KUKA KRL program: EPS_2_251719_MHSUMNERSTREET_A_20251210010858.src

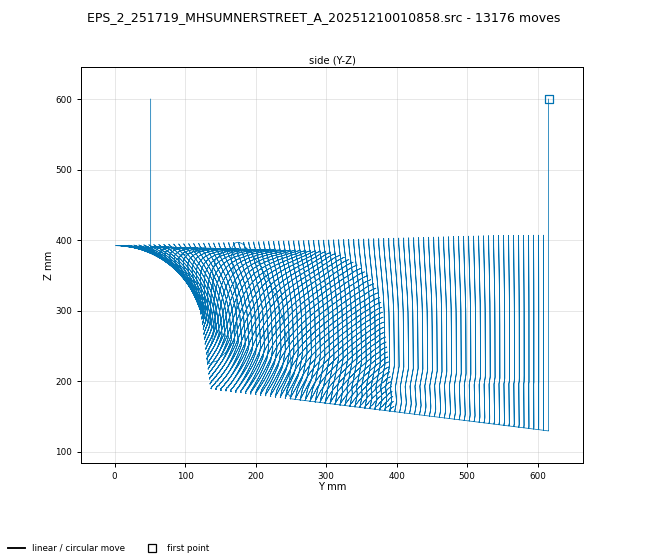
[picture p0: tool path of EPS_2_251719_MHSUMNERSTREET_A_20251210010858.src, 13176 of 13178 moves have a stored position in this frame; points joined in program order, loops and branches not executed]
&ACCESS RVP
&REL 4
&COMMENT QRS 19112012
&PARAM EDITMASK = *
DEF PART()
EXT BAS (BAS_COMMAND :IN,REAL :IN )
INT I
BAS (#INITMOV,0 )

;KUKA QRS Post kuka4.cps  Date:22-06-2017 !

File_ID=2952

QRS_PRE_INIT()

;Init var - Until changes are made in qrs_pre_init
Outlet_Square_prg=0
Inlet_1_Square_prg=0
Inlet_2_Square_prg=0
Inlet_3_Square_prg=0
Inlet_4_Square_prg=0
Inlet_5_Square_prg=0

Outlet_1={X 0.000, Y 546.330, Z 306.500, B 0.000, E1 0.000 }
Inlet_1={X 0.000, Y 567.240, Z 281.500, B 0.000, E1 180.000 }
Outlet_1_type=201
Inlet_1_type=0
;QRS#1=Sidecore dimensions
;QRS#2=200-8" PVC SDR 35
;QRS#3=DeadEnd 201
;QRS#4=
;QRS#5=
;QRS#6=
;QRS#7=
;QRS#8=
;QRS#9=12-08 PSX
;QRS#10=

;QRS#11=
;QRS#12=
;QRS#13=
;QRS#14=
;QRS#15=
;QRS#16=1220x127x686 2,25'
;QRS#17=EPS Height
;QRS#18=407
;QRS#19=*
;QRS#20= UPDATED VERSION 22-06-2017
;QRS#21=*
Outlet_Square=0100
Inlet_1_Square=00
Inlet_2_Square=0
Inlet_3_Square=0
Inlet_4_Square=0
Inlet_5_Square=0
Mill_Square=1
Outlet_Square_Prg=204
Inlet_1_Square_prg=0

QRS_INIT()

$ADVANCE=5

; T1
PTP {E1 173.614,E2 173.614}
PTP {X 0,Y 615.484,A -85,B 0,C 180,E1 173.614,E2 173.614,E3 0,E4 0,E5 0,E6 0}
QRS_SPEED_INIT()
LIN {X 0,Y 615.484,Z 600,A -85,B 0,C 180,E1 173.614,E2 173.614,E3 0,E4 0,E5 0,E6 0} C_VEL
LIN {X 0,Y 615.484,Z 139.376,A -85,B 0,C 180,E1 173.614,E2 173.614} C_VEL
LIN {X 0,Y 615.484,Z 131.194,A -85,B 0,C 180,E1 173.614,E2 173.614} C_VEL
LIN {X 0,Y 615.473,Z 129.194,A -85,B 0,C 180,E1 173.428,E2 173.428} C_VEL
LIN {X 0,Y 615.496,Z 129.181,A -85,B 0,C 180,E1 170.802,E2 170.802} C_VEL
LIN {X 0,Y 615.487,Z 129.196,A -85,B 0,C 180,E1 168.14,E2 168.14} C_VEL
LIN {X 0,Y 615.472,Z 129.19,A -85,B 0,C 180,E1 165.451,E2 165.451} C_VEL
LIN {X 0,Y 615.485,Z 129.186,A -85,B 0,C 180,E1 162.73,E2 162.73} C_VEL
LIN {X 0,Y 615.482,Z 129.198,A -85,B 0,C 180,E1 159.967,E2 159.967} C_VEL
LIN {X 0,Y 615.487,Z 129.183,A -85,B 0,C 180,E1 157.156,E2 157.156} C_VEL
LIN {X 0,Y 615.498,Z 129.2,A -85,B 0,C 180,E1 154.285,E2 154.285} C_VEL
LIN {X 0,Y 615.486,Z 129.183,A -85,B 0,C 180,E1 151.342,E2 151.342} C_VEL
LIN {X 0,Y 615.48,Z 129.19,A -85,B 0,C 180,E1 148.914,E2 148.914} C_VEL
LIN {X 0,Y 615.496,Z 129.199,A -85,B 0,C 180,E1 146.464,E2 146.464} C_VEL
LIN {X 0,Y 615.483,Z 129.184,A -85,B 0,C 180,E1 143.575,E2 143.575} C_VEL
LIN {X 0,Y 615.484,Z 129.194,A -85,B 0,C 180,E1 140.938,E2 140.938} C_VEL
LIN {X 0,Y 615.485,Z 129.197,A -85,B 0,C 180,E1 138.527,E2 138.527} C_VEL
LIN {X 0,Y 615.49,Z 129.182,A -85,B 0,C 180,E1 135.851,E2 135.851} C_VEL
LIN {X 0,Y 615.488,Z 129.196,A -85,B 0,C 180,E1 133.048,E2 133.048} C_VEL
LIN {X 0,Y 615.479,Z 129.194,A -85,B 0,C 180,E1 130.607,E2 130.607} C_VEL
LIN {X 0,Y 615.482,Z 129.184,A -85,B 0,C 180,E1 128.012,E2 128.012} C_VEL
LIN {X 0,Y 615.481,Z 129.188,A -85,B 0,C 180,E1 125.616,E2 125.616} C_VEL
LIN {X 0,Y 615.484,Z 129.199,A -85,B 0,C 180,E1 123.236,E2 123.236} C_VEL
LIN {X 0,Y 615.478,Z 129.196,A -85,B 0,C 180,E1 120.92,E2 120.92} C_VEL
LIN {X 0,Y 615.483,Z 129.185,A -85,B 0,C 180,E1 118.45,E2 118.45} C_VEL
LIN {X 0,Y 615.484,Z 129.195,A -85,B 0,C 180,E1 115.569,E2 115.569} C_VEL
LIN {X 0,Y 615.475,Z 129.19,A -85,B 0,C 180,E1 112.845,E2 112.845} C_VEL
LIN {X 0,Y 615.49,Z 129.183,A -85,B 0,C 180,E1 110.559,E2 110.559} C_VEL
LIN {X 0,Y 615.479,Z 129.191,A -85,B 0,C 180,E1 107.957,E2 107.957} C_VEL
LIN {X 0,Y 615.479,Z 129.193,A -85,B 0,C 180,E1 105.226,E2 105.226} C_VEL
LIN {X 0,Y 615.491,Z 129.182,A -85,B 0,C 180,E1 102.53,E2 102.53} C_VEL
LIN {X 0,Y 615.491,Z 129.198,A -85,B 0,C 180,E1 99.862,E2 99.862} C_VEL
LIN {X 0,Y 615.477,Z 129.189,A -85,B 0,C 180,E1 97.216,E2 97.216} C_VEL
LIN {X 0,Y 615.482,Z 129.186,A -85,B 0,C 180,E1 94.585,E2 94.585} C_VEL
LIN {X 0,Y 615.499,Z 129.2,A -85,B 0,C 180,E1 91.963,E2 91.963} C_VEL
LIN {X 0,Y 615.481,Z 129.187,A -85,B 0,C 180,E1 89.346,E2 89.346} C_VEL
LIN {X 0,Y 615.479,Z 129.187,A -85,B 0,C 180,E1 86.727,E2 86.727} C_VEL
LIN {X 0,Y 615.496,Z 129.199,A -85,B 0,C 180,E1 84.102,E2 84.102} C_VEL
LIN {X 0,Y 615.485,Z 129.185,A -85,B 0,C 180,E1 81.463,E2 81.463} C_VEL
LIN {X 0,Y 615.477,Z 129.19,A -85,B 0,C 180,E1 78.807,E2 78.807} C_VEL
LIN {X 0,Y 615.482,Z 129.194,A -85,B 0,C 180,E1 76.067,E2 76.067} C_VEL
LIN {X 0,Y 615.487,Z 129.183,A -85,B 0,C 180,E1 73.414,E2 73.414} C_VEL
LIN {X 0,Y 615.484,Z 129.198,A -85,B 0,C 180,E1 70.662,E2 70.662} C_VEL
LIN {X 0,Y 615.479,Z 129.186,A -85,B 0,C 180,E1 67.864,E2 67.864} C_VEL
LIN {X 0,Y 615.488,Z 129.183,A -85,B 0,C 180,E1 65.728,E2 65.728} C_VEL
LIN {X 0,Y 615.484,Z 129.2,A -85,B 0,C 180,E1 62.823,E2 62.823} C_VEL
LIN {X 0,Y 615.499,Z 129.18,A -85,B 0,C 180,E1 59.841,E2 59.841} C_VEL
LIN {X 0,Y 615.478,Z 129.187,A -85,B 0,C 180,E1 57.542,E2 57.542} C_VEL
LIN {X 0,Y 615.477,Z 129.196,A -85,B 0,C 180,E1 55.185,E2 55.185} C_VEL
LIN {X 0,Y 615.486,Z 129.195,A -85,B 0,C 180,E1 52.758,E2 52.758} C_VEL
LIN {X 0,Y 615.485,Z 129.184,A -85,B 0,C 180,E1 49.911,E2 49.911} C_VEL
LIN {X 0,Y 615.488,Z 129.196,A -85,B 0,C 180,E1 46.952,E2 46.952} C_VEL
LIN {X 0,Y 615.481,Z 129.185,A -85,B 0,C 180,E1 43.997,E2 43.997} C_VEL
LIN {X 0,Y 615.485,Z 129.197,A -85,B 0,C 180,E1 41.473,E2 41.473} C_VEL
LIN {X 0,Y 615.481,Z 129.191,A -85,B 0,C 180,E1 38.904,E2 38.904} C_VEL
LIN {X 0,Y 615.483,Z 129.184,A -85,B 0,C 180,E1 36.425,E2 36.425} C_VEL
LIN {X 0,Y 615.496,Z 129.199,A -85,B 0,C 180,E1 33.536,E2 33.536} C_VEL
LIN {X 0,Y 615.484,Z 129.186,A -85,B 0,C 180,E1 30.919,E2 30.919} C_VEL
LIN {X 0,Y 615.48,Z 129.185,A -85,B 0,C 180,E1 28.45,E2 28.45} C_VEL
LIN {X 0,Y 615.488,Z 129.198,A -85,B 0,C 180,E1 25.57,E2 25.57} C_VEL
LIN {X 0,Y 615.487,Z 129.183,A -85,B 0,C 180,E1 22.844,E2 22.844} C_VEL
LIN {X 0,Y 615.482,Z 129.198,A -85,B 0,C 180,E1 20.033,E2 20.033} C_VEL
LIN {X 0,Y 615.481,Z 129.187,A -85,B 0,C 180,E1 17.27,E2 17.27} C_VEL
LIN {X 0,Y 615.472,Z 129.19,A -85,B 0,C 180,E1 14.549,E2 14.549} C_VEL
LIN {X 0,Y 615.487,Z 129.196,A -85,B 0,C 180,E1 11.86,E2 11.86} C_VEL
LIN {X 0,Y 615.496,Z 129.181,A -85,B 0,C 180,E1 9.198,E2 9.198} C_VEL
LIN {X 0,Y 615.474,Z 129.195,A -85,B 0,C 180,E1 6.556,E2 6.556} C_VEL
LIN {X 0,Y 615.484,Z 129.192,A -85,B 0,C 180,E1 3.928,E2 3.928} C_VEL
LIN {X 0,Y 615.487,Z 129.183,A -85,B 0,C 180,E1 1.308,E2 1.308} C_VEL
LIN {X 0,Y 615.479,Z 129.195,A -85,B 0,C 180,E1 -1.309,E2 -1.309} C_VEL
LIN {X 0,Y 615.483,Z 129.191,A -85,B 0,C 180,E1 -3.929,E2 -3.929} C_VEL
LIN {X 0,Y 615.48,Z 129.185,A -85,B 0,C 180,E1 -6.577,E2 -6.577} C_VEL
LIN {X 0,Y 615.485,Z 129.197,A -85,B 0,C 180,E1 -9.199,E2 -9.199} C_VEL
LIN {X 0,Y 615.485,Z 129.187,A -85,B 0,C 180,E1 -11.861,E2 -11.861} C_VEL
LIN {X 0,Y 615.473,Z 129.188,A -85,B 0,C 180,E1 -14.55,E2 -14.55} C_VEL
LIN {X 0,Y 615.491,Z 129.198,A -85,B 0,C 180,E1 -17.271,E2 -17.271} C_VEL
LIN {X 0,Y 615.486,Z 129.183,A -85,B 0,C 180,E1 -20.033,E2 -20.033} C_VEL
LIN {X 0,Y 615.48,Z 129.199,A -85,B 0,C 180,E1 -22.845,E2 -22.845} C_VEL
LIN {X 0,Y 615.495,Z 129.182,A -85,B 0,C 180,E1 -25.716,E2 -25.716} C_VEL
LIN {X 0,Y 615.473,Z 129.193,A -85,B 0,C 180,E1 -28.449,E2 -28.449} C_VEL
LIN {X 0,Y 615.486,Z 129.193,A -85,B 0,C 180,E1 -31.087,E2 -31.087} C_VEL
LIN {X 0,Y 615.471,Z 129.188,A -85,B 0,C 180,E1 -34.023,E2 -34.023} C_VEL
LIN {X 0,Y 615.48,Z 129.197,A -85,B 0,C 180,E1 -36.426,E2 -36.426} C_VEL
LIN {X 0,Y 615.485,Z 129.189,A -85,B 0,C 180,E1 -39.063,E2 -39.063} C_VEL
LIN {X 0,Y 615.484,Z 129.184,A -85,B 0,C 180,E1 -41.474,E2 -41.474} C_VEL
LIN {X 0,Y 615.475,Z 129.196,A -85,B 0,C 180,E1 -44.151,E2 -44.151} C_VEL
LIN {X 0,Y 615.486,Z 129.187,A -85,B 0,C 180,E1 -46.953,E2 -46.953} C_VEL
LIN {X 0,Y 615.477,Z 129.185,A -85,B 0,C 180,E1 -49.393,E2 -49.393} C_VEL
LIN {X 0,Y 615.478,Z 129.196,A -85,B 0,C 180,E1 -51.99,E2 -51.99} C_VEL
LIN {X 0,Y 615.489,Z 129.195,A -85,B 0,C 180,E1 -54.385,E2 -54.385} C_VEL
LIN {X 0,Y 615.486,Z 129.186,A -85,B 0,C 180,E1 -56.764,E2 -56.764} C_VEL
LIN {X 0,Y 615.479,Z 129.185,A -85,B 0,C 180,E1 -59.08,E2 -59.08} C_VEL
LIN {X 0,Y 615.471,Z 129.193,A -85,B 0,C 180,E1 -61.553,E2 -61.553} C_VEL
LIN {X 0,Y 615.487,Z 129.188,A -85,B 0,C 180,E1 -64.432,E2 -64.432} C_VEL
LIN {X 0,Y 615.497,Z 129.361,A -85,B 0,C 180,E1 -65.958,E2 -65.958} C_VEL
LIN {X 0,Y 615.498,Z 144.439,A -85,B 0,C 180,E1 -68.569,E2 -68.569} C_VEL
LIN {X 0,Y 615.482,Z 161.223,A -85,B 0,C 180,E1 -71.398,E2 -71.398} C_VEL
LIN {X 0,Y 615.496,Z 178.498,A -85,B 0,C 180,E1 -74.265,E2 -74.265} C_VEL
LIN {X 0,Y 615.469,Z 195.732,A -85,B 0,C 180,E1 -77.071,E2 -77.071} C_VEL
LIN {X 0,Y 615.464,Z 197.255,A -85,B 0,C 180,E1 -77.155,E2 -77.155} C_VEL
LIN {X 0,Y 615.498,Z 302.835,A -85,B 0,C 180,E1 -78.411,E2 -78.411} C_VEL
LIN {X 0,Y 615.499,Z 315.346,A -85,B 0,C 180,E1 -78.682,E2 -78.682} C_VEL
LIN {X 0,Y 615.496,Z 328.502,A -85,B 0,C 180,E1 -79.109,E2 -79.109} C_VEL
LIN {X 0,Y 615.487,Z 340.479,A -85,B 0,C 180,E1 -79.64,E2 -79.64} C_VEL
LIN {X 0,Y 615.493,Z 351.996,A -85,B 0,C 180,E1 -80.304,E2 -80.304} C_VEL
LIN {X 0,Y 615.499,Z 362.342,A -85,B 0,C 180,E1 -81.05,E2 -81.05} C_VEL
LIN {X 0,Y 615.497,Z 370.813,A -85,B 0,C 180,E1 -81.794,E2 -81.794} C_VEL
LIN {X 0,Y 615.498,Z 378.607,A -85,B 0,C 180,E1 -82.62,E2 -82.62} C_VEL
LIN {X 0,Y 615.496,Z 386.203,A -85,B 0,C 180,E1 -83.608,E2 -83.608} C_VEL
LIN {X 0,Y 615.498,Z 393.205,A -85,B 0,C 180,E1 -84.759,E2 -84.759} C_VEL
LIN {X 0,Y 615.493,Z 397.852,A -85,B 0,C 180,E1 -85.744,E2 -85.744} C_VEL
LIN {X 0,Y 615.494,Z 401.399,A -85,B 0,C 180,E1 -86.727,E2 -86.727} C_VEL
LIN {X 0,Y 615.497,Z 403.233,A -85,B 0,C 180,E1 -87.382,E2 -87.382} C_VEL
LIN {X 0,Y 615.5,Z 404.607,A -85,B 0,C 180,E1 -88.037,E2 -88.037} C_VEL
LIN {X 0,Y 615.496,Z 406.173,A -85,B 0,C 180,E1 -89.346,E2 -89.346} C_VEL
LIN {X 0,Y 615.494,Z 406.389,A -85,B 0,C 180,E1 -90,E2 -90} C_VEL
LIN {X 0,Y 615.495,Z 405.58,A -85,B 0,C 180,E1 -91.309,E2 -91.309} C_VEL
LIN {X 0,Y 615.5,Z 404.607,A -85,B 0,C 180,E1 -91.963,E2 -91.963} C_VEL
LIN {X 0,Y 615.497,Z 403.233,A -85,B 0,C 180,E1 -92.618,E2 -92.618} C_VEL
LIN {X 0,Y 615.496,Z 400.35,A -85,B 0,C 180,E1 -93.601,E2 -93.601} C_VEL
LIN {X 0,Y 615.498,Z 396.442,A -85,B 0,C 180,E1 -94.584,E2 -94.584} C_VEL
LIN {X 0,Y 615.499,Z 391.405,A -85,B 0,C 180,E1 -95.57,E2 -95.57} C_VEL
LIN {X 0,Y 615.497,Z 384.87,A -85,B 0,C 180,E1 -96.583,E2 -96.583} C_VEL
LIN {X 0,Y 615.497,Z 377.134,A -85,B 0,C 180,E1 -97.545,E2 -97.545} C_VEL
LIN {X 0,Y 615.498,Z 369.046,A -85,B 0,C 180,E1 -98.371,E2 -98.371} C_VEL
LIN {X 0,Y 615.499,Z 359.169,A -85,B 0,C 180,E1 -99.199,E2 -99.199} C_VEL
LIN {X 0,Y 615.487,Z 347.983,A -85,B 0,C 180,E1 -99.945,E2 -99.945} C_VEL
LIN {X 0,Y 615.492,Z 337.024,A -85,B 0,C 180,E1 -100.527,E2 -100.527} C_VEL
LIN {X 0,Y 615.499,Z 324.42,A -85,B 0,C 180,E1 -101.042,E2 -101.042} C_VEL
LIN {X 0,Y 615.499,Z 312.068,A -85,B 0,C 180,E1 -101.401,E2 -101.401} C_VEL
LIN {X 0,Y 615.499,Z 298.472,A -85,B 0,C 180,E1 -101.652,E2 -101.652} C_VEL
LIN {X 0,Y 615.465,Z 196.548,A -85,B 0,C 180,E1 -102.866,E2 -102.866} C_VEL
LIN {X 0,Y 615.478,Z 194.988,A -85,B 0,C 180,E1 -103.033,E2 -103.033} C_VEL
LIN {X 0,Y 615.493,Z 177.465,A -85,B 0,C 180,E1 -105.905,E2 -105.905} C_VEL
LIN {X 0,Y 615.49,Z 159.928,A -85,B 0,C 180,E1 -108.818,E2 -108.818} C_VEL
LIN {X 0,Y 615.484,Z 143.406,A -85,B 0,C 180,E1 -111.608,E2 -111.608} C_VEL
LIN {X 0,Y 615.497,Z 129.361,A -85,B 0,C 180,E1 -114.042,E2 -114.042} C_VEL
LIN {X 0,Y 615.47,Z 129.194,A -85,B 0,C 180,E1 -116.445,E2 -116.445} C_VEL
LIN {X 0,Y 615.469,Z 129.19,A -85,B 0,C 180,E1 -118.659,E2 -118.659} C_VEL
LIN {X 0,Y 615.485,Z 129.184,A -85,B 0,C 180,E1 -121.085,E2 -121.085} C_VEL
LIN {X 0,Y 615.483,Z 129.198,A -85,B 0,C 180,E1 -124.022,E2 -124.022} C_VEL
LIN {X 0,Y 615.488,Z 129.183,A -85,B 0,C 180,E1 -126.936,E2 -126.936} C_VEL
LIN {X 0,Y 615.496,Z 129.199,A -85,B 0,C 180,E1 -129.749,E2 -129.749} C_VEL
LIN {X 0,Y 615.47,Z 129.188,A -85,B 0,C 180,E1 -132.354,E2 -132.354} C_VEL
LIN {X 0,Y 615.486,Z 129.188,A -85,B 0,C 180,E1 -135.068,E2 -135.068} C_VEL
LIN {X 0,Y 615.482,Z 129.199,A -85,B 0,C 180,E1 -137.646,E2 -137.646} C_VEL
LIN {X 0,Y 615.474,Z 129.186,A -85,B 0,C 180,E1 -140.248,E2 -140.248} C_VEL
LIN {X 0,Y 615.486,Z 129.193,A -85,B 0,C 180,E1 -143.063,E2 -143.063} C_VEL
LIN {X 0,Y 615.491,Z 129.202,A -85,B 0,C 180,E1 -145.298,E2 -145.298} C_VEL
LIN {X 0,Y 615.472,Z 129.193,A -85,B 0,C 180,E1 -147.671,E2 -147.671} C_VEL
LIN {X 0,Y 615.487,Z 129.183,A -85,B 0,C 180,E1 -150.204,E2 -150.204} C_VEL
LIN {X 0,Y 615.491,Z 129.197,A -85,B 0,C 180,E1 -152.953,E2 -152.953} C_VEL
LIN {X 0,Y 615.472,Z 129.188,A -85,B 0,C 180,E1 -155.727,E2 -155.727} C_VEL
LIN {X 0,Y 615.484,Z 129.191,A -85,B 0,C 180,E1 -158.568,E2 -158.568} C_VEL
LIN {X 0,Y 615.471,Z 129.191,A -85,B 0,C 180,E1 -161.398,E2 -161.398} C_VEL
LIN {X 0,Y 615.491,Z 129.184,A -85,B 0,C 180,E1 -164.095,E2 -164.095} C_VEL
LIN {X 0,Y 615.494,Z 129.199,A -85,B 0,C 180,E1 -166.799,E2 -166.799} C_VEL
LIN {X 0,Y 615.477,Z 129.186,A -85,B 0,C 180,E1 -169.473,E2 -169.473} C_VEL
LIN {X 0,Y 615.483,Z 129.19,A -85,B 0,C 180,E1 -172.124,E2 -172.124} C_VEL
LIN {X 0,Y 615.481,Z 129.196,A -85,B 0,C 180,E1 -174.758,E2 -174.758} C_VEL
LIN {X 0,Y 615.484,Z 129.184,A -85,B 0,C 180,E1 -177.382,E2 -177.382} C_VEL
LIN {X 0,Y 615.483,Z 129.192,A -85,B 0,C 180,E1 -180,E2 -180} C_VEL
LIN {X 0,Y 615.478,Z 129.195,A -85,B 0,C 180,E1 -182.618,E2 -182.618} C_VEL
LIN {X 0,Y 615.49,Z 129.182,A -85,B 0,C 180,E1 -185.241,E2 -185.241} C_VEL
LIN {X 0,Y 615.473,Z 129.194,A -85,B 0,C 180,E1 -186.572,E2 -186.572} C_VEL
LIN {X 0,Y 614.807,Z 129.333,A -85,B 0,C 180,E1 -187.118,E2 -187.118} C_VEL
LIN {X 0,Y 611.985,Z 129.755,A -85,B 0,C 180,E1 -188.004,E2 -188.004} C_VEL
LIN {X 0,Y 609.596,Z 130.06,A -85,B 0,C 180,E1 -188.717,E2 -188.717} C_VEL
LIN {X 0,Y 608.556,Z 130.176,A -85,B 0,C 180,E1 -189.266,E2 -189.266} C_VEL
LIN {X 0,Y 608.464,Z 130.187,A -85,B 0,C 180,E1 -189.452,E2 -189.452} C_VEL
LIN {X 0,Y 608.46,Z 130.196,A -85,B 0,C 180,E1 -191.999,E2 -191.999} C_VEL
LIN {X 0,Y 608.467,Z 130.187,A -85,B 0,C 180,E1 -194.72,E2 -194.72} C_VEL
LIN {X 0,Y 608.454,Z 130.191,A -85,B 0,C 180,E1 -197.476,E2 -197.476} C_VEL
LIN {X 0,Y 608.456,Z 130.191,A -85,B 0,C 180,E1 -200.274,E2 -200.274} C_VEL
LIN {X 0,Y 608.451,Z 130.189,A -85,B 0,C 180,E1 -203.124,E2 -203.124} C_VEL
LIN {X 0,Y 608.449,Z 130.192,A -85,B 0,C 180,E1 -206.035,E2 -206.035} C_VEL
LIN {X 0,Y 608.469,Z 130.185,A -85,B 0,C 180,E1 -208.62,E2 -208.62} C_VEL
LIN {X 0,Y 608.472,Z 130.192,A -85,B 0,C 180,E1 -211.316,E2 -211.316} C_VEL
LIN {X 0,Y 608.475,Z 130.191,A -85,B 0,C 180,E1 -213.736,E2 -213.736} C_VEL
LIN {X 0,Y 608.471,Z 130.186,A -85,B 0,C 180,E1 -216.09,E2 -216.09} C_VEL
LIN {X 0,Y 608.463,Z 130.187,A -85,B 0,C 180,E1 -218.588,E2 -218.588} C_VEL
LIN {X 0,Y 608.46,Z 130.196,A -85,B 0,C 180,E1 -221.343,E2 -221.343} C_VEL
LIN {X 0,Y 608.458,Z 130.187,A -85,B 0,C 180,E1 -224.265,E2 -224.265} C_VEL
LIN {X 0,Y 608.453,Z 130.196,A -85,B 0,C 180,E1 -227.041,E2 -227.041} C_VEL
LIN {X 0,Y 608.447,Z 130.19,A -85,B 0,C 180,E1 -229.697,E2 -229.697} C_VEL
LIN {X 0,Y 608.467,Z 130.187,A -85,B 0,C 180,E1 -232.254,E2 -232.254} C_VEL
LIN {X 0,Y 608.473,Z 130.192,A -85,B 0,C 180,E1 -235.091,E2 -235.091} C_VEL
LIN {X 0,Y 608.463,Z 130.186,A -85,B 0,C 180,E1 -237.906,E2 -237.906} C_VEL
LIN {X 0,Y 608.465,Z 130.188,A -85,B 0,C 180,E1 -240.221,E2 -240.221} C_VEL
LIN {X 0,Y 608.477,Z 130.194,A -85,B 0,C 180,E1 -242.792,E2 -242.792} C_VEL
LIN {X 0,Y 608.452,Z 130.188,A -85,B 0,C 180,E1 -245.429,E2 -245.429} C_VEL
LIN {X 0,Y 608.473,Z 130.191,A -85,B 0,C 180,E1 -248.309,E2 -248.309} C_VEL
LIN {X 0,Y 608.471,Z 130.186,A -85,B 0,C 180,E1 -251.283,E2 -251.283} C_VEL
LIN {X 0,Y 608.458,Z 130.19,A -85,B 0,C 180,E1 -253.906,E2 -253.906} C_VEL
LIN {X 0,Y 608.456,Z 130.193,A -85,B 0,C 180,E1 -256.644,E2 -256.644} C_VEL
LIN {X 0,Y 608.464,Z 130.186,A -85,B 0,C 180,E1 -259.35,E2 -259.35} C_VEL
LIN {X 0,Y 608.477,Z 130.192,A -85,B 0,C 180,E1 -262.033,E2 -262.033} C_VEL
LIN {X 0,Y 608.46,Z 130.189,A -85,B 0,C 180,E1 -264.698,E2 -264.698} C_VEL
LIN {X 0,Y 608.472,Z 130.186,A -85,B 0,C 180,E1 -267.352,E2 -267.352} C_VEL
LIN {X 0,Y 608.477,Z 130.195,A -85,B 0,C 180,E1 -270,E2 -270} C_VEL
LIN {X 0,Y 608.472,Z 130.186,A -85,B 0,C 180,E1 -272.648,E2 -272.648} C_VEL
LIN {X 0,Y 608.46,Z 130.189,A -85,B 0,C 180,E1 -275.302,E2 -275.302} C_VEL
LIN {X 0,Y 608.477,Z 130.192,A -85,B 0,C 180,E1 -277.967,E2 -277.967} C_VEL
LIN {X 0,Y 608.467,Z 130.186,A -85,B 0,C 180,E1 -280.957,E2 -280.957} C_VEL
LIN {X 0,Y 608.455,Z 130.193,A -85,B 0,C 180,E1 -283.356,E2 -283.356} C_VEL
LIN {X 0,Y 608.456,Z 130.19,A -85,B 0,C 180,E1 -286.094,E2 -286.094} C_VEL
LIN {X 0,Y 608.455,Z 130.189,A -85,B 0,C 180,E1 -288.869,E2 -288.869} C_VEL
LIN {X 0,Y 608.473,Z 130.191,A -85,B 0,C 180,E1 -291.691,E2 -291.691} C_VEL
LIN {X 0,Y 608.45,Z 130.188,A -85,B 0,C 180,E1 -294.571,E2 -294.571} C_VEL
LIN {X 0,Y 608.477,Z 130.194,A -85,B 0,C 180,E1 -297.208,E2 -297.208} C_VEL
LIN {X 0,Y 608.468,Z 130.186,A -85,B 0,C 180,E1 -299.972,E2 -299.972} C_VEL
LIN {X 0,Y 608.454,Z 130.189,A -85,B 0,C 180,E1 -302.522,E2 -302.522} C_VEL
LIN {X 0,Y 608.437,Z 130.196,A -85,B 0,C 180,E1 -305.278,E2 -305.278} C_VEL
LIN {X 0,Y 608.468,Z 130.186,A -85,B 0,C 180,E1 -307.746,E2 -307.746} C_VEL
LIN {X 0,Y 608.448,Z 130.19,A -85,B 0,C 180,E1 -310.329,E2 -310.329} C_VEL
LIN {X 0,Y 608.453,Z 130.196,A -85,B 0,C 180,E1 -312.959,E2 -312.959} C_VEL
LIN {X 0,Y 608.458,Z 130.187,A -85,B 0,C 180,E1 -315.735,E2 -315.735} C_VEL
LIN {X 0,Y 608.46,Z 130.196,A -85,B 0,C 180,E1 -318.657,E2 -318.657} C_VEL
LIN {X 0,Y 608.463,Z 130.187,A -85,B 0,C 180,E1 -321.412,E2 -321.412} C_VEL
LIN {X 0,Y 608.471,Z 130.187,A -85,B 0,C 180,E1 -323.951,E2 -323.951} C_VEL
LIN {X 0,Y 608.467,Z 130.193,A -85,B 0,C 180,E1 -326.33,E2 -326.33} C_VEL
LIN {X 0,Y 608.472,Z 130.191,A -85,B 0,C 180,E1 -328.727,E2 -328.727} C_VEL
LIN {X 0,Y 608.471,Z 130.185,A -85,B 0,C 180,E1 -331.379,E2 -331.379} C_VEL
LIN {X 0,Y 608.477,Z 130.195,A -85,B 0,C 180,E1 -334.277,E2 -334.277} C_VEL
LIN {X 0,Y 608.451,Z 130.189,A -85,B 0,C 180,E1 -336.876,E2 -336.876} C_VEL
LIN {X 0,Y 608.456,Z 130.191,A -85,B 0,C 180,E1 -339.726,E2 -339.726} C_VEL
LIN {X 0,Y 608.452,Z 130.191,A -85,B 0,C 180,E1 -342.524,E2 -342.524} C_VEL
LIN {X 0,Y 608.467,Z 130.187,A -85,B 0,C 180,E1 -345.28,E2 -345.28} C_VEL
LIN {X 0,Y 608.46,Z 130.196,A -85,B 0,C 180,E1 -348.001,E2 -348.001} C_VEL
LIN {X 0,Y 608.477,Z 130.184,A -85,B 0,C 180,E1 -350.695,E2 -350.695} C_VEL
LIN {X 0,Y 608.452,Z 130.191,A -85,B 0,C 180,E1 -353.385,E2 -353.385} C_VEL
LIN {X 0,Y 608.452,Z 130.193,A -85,B 0,C 180,E1 -356.026,E2 -356.026} C_VEL
LIN {X 0,Y 608.47,Z 130.185,A -85,B 0,C 180,E1 -358.677,E2 -358.677} C_VEL
LIN {X 0,Y 608.463,Z 130.192,A -85,B 0,C 180,E1 -361.324,E2 -361.324} C_VEL
LIN {X 0,Y 608.452,Z 130.191,A -85,B 0,C 180,E1 -363.974,E2 -363.974} C_VEL
LIN {X 0,Y 608.474,Z 130.185,A -85,B 0,C 180,E1 -366.633,E2 -366.633} C_VEL
LIN {X 0,Y 608.469,Z 130.195,A -85,B 0,C 180,E1 -369.306,E2 -369.306} C_VEL
LIN {X 0,Y 608.458,Z 130.188,A -85,B 0,C 180,E1 -372,E2 -372} C_VEL
LIN {X 0,Y 608.467,Z 130.188,A -85,B 0,C 180,E1 -374.721,E2 -374.721} C_VEL
LIN {X 0,Y 608.457,Z 130.192,A -85,B 0,C 180,E1 -377.477,E2 -377.477} C_VEL
LIN {X 0,Y 608.456,Z 130.187,A -85,B 0,C 180,E1 -380.275,E2 -380.275} C_VEL
LIN {X 0,Y 608.456,Z 130.189,A -85,B 0,C 180,E1 -382.477,E2 -382.477} C_VEL
LIN {X 0,Y 608.453,Z 130.192,A -85,B 0,C 180,E1 -385.301,E2 -385.301} C_VEL
LIN {X 0,Y 608.448,Z 130.189,A -85,B 0,C 180,E1 -387.518,E2 -387.518} C_VEL
LIN {X 0,Y 608.463,Z 130.186,A -85,B 0,C 180,E1 -389.972,E2 -389.972} C_VEL
LIN {X 0,Y 608.454,Z 130.194,A -85,B 0,C 180,E1 -392.522,E2 -392.522} C_VEL
LIN {X 0,Y 608.448,Z 130.19,A -85,B 0,C 180,E1 -395.278,E2 -395.278} C_VEL
LIN {X 0,Y 608.46,Z 130.187,A -85,B 0,C 180,E1 -397.747,E2 -397.747} C_VEL
LIN {X 0,Y 608.445,Z 130.195,A -85,B 0,C 180,E1 -400.329,E2 -400.329} C_VEL
LIN {X 0,Y 608.481,Z 130.184,A -85,B 0,C 180,E1 -403.311,E2 -403.311} C_VEL
LIN {X 0,Y 608.46,Z 130.192,A -85,B 0,C 180,E1 -406.13,E2 -406.13} C_VEL
LIN {X 0,Y 608.458,Z 130.189,A -85,B 0,C 180,E1 -408.824,E2 -408.824} C_VEL
LIN {X 0,Y 608.47,Z 130.186,A -85,B 0,C 180,E1 -411.413,E2 -411.413} C_VEL
LIN {X 0,Y 608.447,Z 130.195,A -85,B 0,C 180,E1 -413.955,E2 -413.955} C_VEL
LIN {X 0,Y 608.467,Z 130.193,A -85,B 0,C 180,E1 -416.33,E2 -416.33} C_VEL
LIN {X 0,Y 608.479,Z 130.186,A -85,B 0,C 180,E1 -418.728,E2 -418.728} C_VEL
LIN {X 0,Y 608.459,Z 130.188,A -85,B 0,C 180,E1 -421.383,E2 -421.383} C_VEL
LIN {X 0,Y 608.44,Z 130.2,A -85,B 0,C 180,E1 -423.965,E2 -423.965} C_VEL
LIN {X 0,Y 608.496,Z 130.349,A -85,B 0,C 180,E1 -425.844,E2 -425.844} C_VEL
LIN {X 0,Y 608.531,Z 144.463,A -85,B 0,C 180,E1 -428.311,E2 -428.311} C_VEL
LIN {X 0,Y 608.51,Z 161.02,A -85,B 0,C 180,E1 -431.132,E2 -431.132} C_VEL
LIN {X 0,Y 608.483,Z 177.577,A -85,B 0,C 180,E1 -433.907,E2 -433.907} C_VEL
LIN {X 0,Y 608.481,Z 194.133,A -85,B 0,C 180,E1 -436.644,E2 -436.644} C_VEL
LIN {X 0,Y 608.461,Z 196.249,A -85,B 0,C 180,E1 -436.962,E2 -436.962} C_VEL
LIN {X 0,Y 608.539,Z 198.731,A -85,B 0,C 180,E1 -437.028,E2 -437.028} C_VEL
LIN {X 0,Y 608.548,Z 302.943,A -85,B 0,C 180,E1 -438.277,E2 -438.277} C_VEL
LIN {X 0,Y 608.548,Z 316.23,A -85,B 0,C 180,E1 -438.572,E2 -438.572} C_VEL
LIN {X 0,Y 608.54,Z 329.391,A -85,B 0,C 180,E1 -439.011,E2 -439.011} C_VEL
LIN {X 0,Y 608.51,Z 340.623,A -85,B 0,C 180,E1 -439.519,E2 -439.519} C_VEL
LIN {X 0,Y 608.482,Z 352.199,A -85,B 0,C 180,E1 -440.191,E2 -440.191} C_VEL
LIN {X 0,Y 608.474,Z 363.647,A -85,B 0,C 180,E1 -441.029,E2 -441.029} C_VEL
LIN {X 0,Y 608.463,Z 372.784,A -85,B 0,C 180,E1 -441.866,E2 -441.866} C_VEL
LIN {X 0,Y 608.466,Z 381.688,A -85,B 0,C 180,E1 -442.867,E2 -442.867} C_VEL
LIN {X 0,Y 608.443,Z 388.85,A -85,B 0,C 180,E1 -443.867,E2 -443.867} C_VEL
LIN {X 0,Y 608.437,Z 395.365,A -85,B 0,C 180,E1 -445.03,E2 -445.03} C_VEL
LIN {X 0,Y 608.435,Z 399.675,A -85,B 0,C 180,E1 -446.026,E2 -446.026} C_VEL
LIN {X 0,Y 608.425,Z 401.957,A -85,B 0,C 180,E1 -446.689,E2 -446.689} C_VEL
LIN {X 0,Y 608.425,Z 403.808,A -85,B 0,C 180,E1 -447.352,E2 -447.352} C_VEL
LIN {X 0,Y 608.445,Z 405.201,A -85,B 0,C 180,E1 -448.014,E2 -448.014} C_VEL
LIN {X 0,Y 608.438,Z 406.783,A -85,B 0,C 180,E1 -449.338,E2 -449.338} C_VEL
LIN {X 0,Y 608.434,Z 406.998,A -85,B 0,C 180,E1 -450,E2 -450} C_VEL
LIN {X 0,Y 608.448,Z 406.184,A -85,B 0,C 180,E1 -451.324,E2 -451.324} C_VEL
LIN {X 0,Y 608.445,Z 405.201,A -85,B 0,C 180,E1 -451.986,E2 -451.986} C_VEL
LIN {X 0,Y 608.425,Z 403.808,A -85,B 0,C 180,E1 -452.648,E2 -452.648} C_VEL
LIN {X 0,Y 608.449,Z 400.896,A -85,B 0,C 180,E1 -453.642,E2 -453.642} C_VEL
LIN {X 0,Y 608.432,Z 396.951,A -85,B 0,C 180,E1 -454.638,E2 -454.638} C_VEL
LIN {X 0,Y 608.451,Z 391.864,A -85,B 0,C 180,E1 -455.634,E2 -455.634} C_VEL
LIN {X 0,Y 608.442,Z 385.472,A -85,B 0,C 180,E1 -456.633,E2 -456.633} C_VEL
LIN {X 0,Y 608.475,Z 377.48,A -85,B 0,C 180,E1 -457.633,E2 -457.633} C_VEL
LIN {X 0,Y 608.487,Z 369.339,A -85,B 0,C 180,E1 -458.468,E2 -458.468} C_VEL
LIN {X 0,Y 608.487,Z 359.396,A -85,B 0,C 180,E1 -459.305,E2 -459.305} C_VEL
LIN {X 0,Y 608.503,Z 348.169,A -85,B 0,C 180,E1 -460.06,E2 -460.06} C_VEL
LIN {X 0,Y 608.518,Z 337.178,A -85,B 0,C 180,E1 -460.649,E2 -460.649} C_VEL
LIN {X 0,Y 608.535,Z 325.708,A -85,B 0,C 180,E1 -461.127,E2 -461.127} C_VEL
LIN {X 0,Y 608.55,Z 313.069,A -85,B 0,C 180,E1 -461.512,E2 -461.512} C_VEL
LIN {X 0,Y 608.563,Z 300.117,A -85,B 0,C 180,E1 -461.765,E2 -461.765} C_VEL
LIN {X 0,Y 608.48,Z 196.578,A -85,B 0,C 180,E1 -463.016,E2 -463.016} C_VEL
LIN {X 0,Y 608.456,Z 195.168,A -85,B 0,C 180,E1 -463.186,E2 -463.186} C_VEL
LIN {X 0,Y 608.498,Z 178.611,A -85,B 0,C 180,E1 -465.921,E2 -465.921} C_VEL
LIN {X 0,Y 608.511,Z 161.856,A -85,B 0,C 180,E1 -468.726,E2 -468.726} C_VEL
LIN {X 0,Y 608.527,Z 145.498,A -85,B 0,C 180,E1 -471.511,E2 -471.511} C_VEL
LIN {X 0,Y 608.552,Z 130.737,A -85,B 0,C 180,E1 -474.072,E2 -474.072} C_VEL
LIN {X 0,Y 608.476,Z 130.256,A -85,B 0,C 180,E1 -474.198,E2 -474.198} C_VEL
LIN {X 0,Y 608.44,Z 130.19,A -85,B 0,C 180,E1 -476.774,E2 -476.774} C_VEL
LIN {X 0,Y 608.475,Z 130.192,A -85,B 0,C 180,E1 -479.779,E2 -479.779} C_VEL
LIN {X 0,Y 608.447,Z 130.19,A -85,B 0,C 180,E1 -482.52,E2 -482.52} C_VEL
LIN {X 0,Y 608.447,Z 130.188,A -85,B 0,C 180,E1 -484.905,E2 -484.905} C_VEL
LIN {X 0,Y 608.465,Z 130.197,A -85,B 0,C 180,E1 -487.746,E2 -487.746} C_VEL
LIN {X 0,Y 608.438,Z 130.191,A -85,B 0,C 180,E1 -490.327,E2 -490.327} C_VEL
LIN {X 0,Y 608.473,Z 130.19,A -85,B 0,C 180,E1 -493.309,E2 -493.309} C_VEL
LIN {X 0,Y 608.46,Z 130.188,A -85,B 0,C 180,E1 -496.129,E2 -496.129} C_VEL
LIN {X 0,Y 608.455,Z 130.189,A -85,B 0,C 180,E1 -498.823,E2 -498.823} C_VEL
LIN {X 0,Y 608.456,Z 130.191,A -85,B 0,C 180,E1 -501.76,E2 -501.76} C_VEL
LIN {X 0,Y 608.443,Z 130.19,A -85,B 0,C 180,E1 -503.954,E2 -503.954} C_VEL
LIN {X 0,Y 608.465,Z 130.186,A -85,B 0,C 180,E1 -506.329,E2 -506.329} C_VEL
LIN {X 0,Y 608.476,Z 130.188,A -85,B 0,C 180,E1 -508.727,E2 -508.727} C_VEL
LIN {X 0,Y 608.466,Z 130.192,A -85,B 0,C 180,E1 -511.38,E2 -511.38} C_VEL
LIN {X 0,Y 608.444,Z 130.188,A -85,B 0,C 180,E1 -513.964,E2 -513.964} C_VEL
LIN {X 0,Y 608.462,Z 130.186,A -85,B 0,C 180,E1 -516.155,E2 -516.155} C_VEL
LIN {X 0,Y 608.45,Z 130.197,A -85,B 0,C 180,E1 -519.018,E2 -519.018} C_VEL
LIN {X 0,Y 608.448,Z 130.188,A -85,B 0,C 180,E1 -521.828,E2 -521.828} C_VEL
LIN {X 0,Y 608.475,Z 130.192,A -85,B 0,C 180,E1 -524.594,E2 -524.594} C_VEL
LIN {X 0,Y 608.469,Z 130.187,A -85,B 0,C 180,E1 -527.323,E2 -527.323} C_VEL
LIN {X 0,Y 608.453,Z 130.189,A -85,B 0,C 180,E1 -530.022,E2 -530.022} C_VEL
LIN {X 0,Y 608.459,Z 130.195,A -85,B 0,C 180,E1 -532.7,E2 -532.7} C_VEL
LIN {X 0,Y 608.451,Z 130.188,A -85,B 0,C 180,E1 -535.362,E2 -535.362} C_VEL
LIN {X 0,Y 608.453,Z 130.191,A -85,B 0,C 180,E1 -538.014,E2 -538.014} C_VEL
LIN {X 0,Y 608.473,Z 130.19,A -85,B 0,C 180,E1 -540.661,E2 -540.661} C_VEL
LIN {X 0,Y 608.477,Z 130.184,A -85,B 0,C 180,E1 -543.31,E2 -543.31} C_VEL
LIN {X 0,Y 608.456,Z 130.193,A -85,B 0,C 180,E1 -545.967,E2 -545.967} C_VEL
LIN {X 0,Y 608.449,Z 130.19,A -85,B 0,C 180,E1 -548.636,E2 -548.636} C_VEL
LIN {X 0,Y 608.464,Z 130.187,A -85,B 0,C 180,E1 -549.452,E2 -549.452} C_VEL
LIN {X 0,Y 607.777,Z 130.28,A -85,B 0,C 180,E1 -550.005,E2 -550.005} C_VEL
LIN {X 0,Y 604.92,Z 130.64,A -85,B 0,C 180,E1 -550.902,E2 -550.902} C_VEL
LIN {X 0,Y 602.519,Z 130.939,A -85,B 0,C 180,E1 -551.623,E2 -551.623} C_VEL
LIN {X 0,Y 601.49,Z 131.063,A -85,B 0,C 180,E1 -552.18,E2 -552.18} C_VEL
LIN {X 0,Y 601.405,Z 131.07,A -85,B 0,C 180,E1 -552.368,E2 -552.368} C_VEL
LIN {X 0,Y 601.425,Z 131.063,A -85,B 0,C 180,E1 -554.897,E2 -554.897} C_VEL
LIN {X 0,Y 601.4,Z 131.072,A -85,B 0,C 180,E1 -557.688,E2 -557.688} C_VEL
LIN {X 0,Y 601.424,Z 131.064,A -85,B 0,C 180,E1 -560.522,E2 -560.522} C_VEL
LIN {X 0,Y 601.418,Z 131.068,A -85,B 0,C 180,E1 -563.41,E2 -563.41} C_VEL
LIN {X 0,Y 601.401,Z 131.066,A -85,B 0,C 180,E1 -566.363,E2 -566.363} C_VEL
LIN {X 0,Y 601.435,Z 131.062,A -85,B 0,C 180,E1 -568.79,E2 -568.79} C_VEL
LIN {X 0,Y 601.408,Z 131.072,A -85,B 0,C 180,E1 -571.726,E2 -571.726} C_VEL
LIN {X 0,Y 601.428,Z 131.063,A -85,B 0,C 180,E1 -574.118,E2 -574.118} C_VEL
LIN {X 0,Y 601.407,Z 131.066,A -85,B 0,C 180,E1 -576.582,E2 -576.582} C_VEL
LIN {X 0,Y 601.433,Z 131.068,A -85,B 0,C 180,E1 -579.536,E2 -579.536} C_VEL
LIN {X 0,Y 601.435,Z 131.064,A -85,B 0,C 180,E1 -582.668,E2 -582.668} C_VEL
LIN {X 0,Y 601.42,Z 131.068,A -85,B 0,C 180,E1 -585.482,E2 -585.482} C_VEL
LIN {X 0,Y 601.421,Z 131.063,A -85,B 0,C 180,E1 -588.407,E2 -588.407} C_VEL
LIN {X 0,Y 601.435,Z 131.069,A -85,B 0,C 180,E1 -590.876,E2 -590.876} C_VEL
LIN {X 0,Y 601.44,Z 131.061,A -85,B 0,C 180,E1 -593.734,E2 -593.734} C_VEL
LIN {X 0,Y 601.424,Z 131.069,A -85,B 0,C 180,E1 -596.687,E2 -596.687} C_VEL
LIN {X 0,Y 601.429,Z 131.068,A -85,B 0,C 180,E1 -599.059,E2 -599.059} C_VEL
LIN {X 0,Y 601.427,Z 131.064,A -85,B 0,C 180,E1 -601.373,E2 -601.373} C_VEL
LIN {X 0,Y 601.399,Z 131.066,A -85,B 0,C 180,E1 -603.636,E2 -603.636} C_VEL
LIN {X 0,Y 601.416,Z 131.074,A -85,B 0,C 180,E1 -606.59,E2 -606.59} C_VEL
LIN {X 0,Y 601.43,Z 131.063,A -85,B 0,C 180,E1 -609.478,E2 -609.478} C_VEL
LIN {X 0,Y 601.393,Z 131.075,A -85,B 0,C 180,E1 -612.312,E2 -612.312} C_VEL
LIN {X 0,Y 601.41,Z 131.076,A -85,B 0,C 180,E1 -614.409,E2 -614.409} C_VEL
LIN {X 0,Y 601.419,Z 131.064,A -85,B 0,C 180,E1 -617.172,E2 -617.172} C_VEL
LIN {X 0,Y 601.436,Z 131.066,A -85,B 0,C 180,E1 -619.905,E2 -619.905} C_VEL
LIN {X 0,Y 601.436,Z 131.066,A -85,B 0,C 180,E1 -622.615,E2 -622.615} C_VEL
LIN {X 0,Y 601.419,Z 131.064,A -85,B 0,C 180,E1 -625.308,E2 -625.308} C_VEL
LIN {X 0,Y 601.436,Z 131.072,A -85,B 0,C 180,E1 -627.991,E2 -627.991} C_VEL
LIN {X 0,Y 601.447,Z 131.062,A -85,B 0,C 180,E1 -630.67,E2 -630.67} C_VEL
LIN {X 0,Y 601.425,Z 131.065,A -85,B 0,C 180,E1 -633.35,E2 -633.35} C_VEL
LIN {X 0,Y 601.42,Z 131.071,A -85,B 0,C 180,E1 -636.037,E2 -636.037} C_VEL
LIN {X 0,Y 601.433,Z 131.062,A -85,B 0,C 180,E1 -638.738,E2 -638.738} C_VEL
LIN {X 0,Y 601.431,Z 131.069,A -85,B 0,C 180,E1 -641.458,E2 -641.458} C_VEL
LIN {X 0,Y 601.417,Z 131.066,A -85,B 0,C 180,E1 -644.205,E2 -644.205} C_VEL
LIN {X 0,Y 601.429,Z 131.065,A -85,B 0,C 180,E1 -646.986,E2 -646.986} C_VEL
LIN {X 0,Y 601.403,Z 131.071,A -85,B 0,C 180,E1 -649.809,E2 -649.809} C_VEL
LIN {X 0,Y 601.412,Z 131.065,A -85,B 0,C 180,E1 -652.606,E2 -652.606} C_VEL
LIN {X 0,Y 601.399,Z 131.07,A -85,B 0,C 180,E1 -654.878,E2 -654.878} C_VEL
LIN {X 0,Y 601.418,Z 131.066,A -85,B 0,C 180,E1 -657.867,E2 -657.867} C_VEL
LIN {X 0,Y 601.445,Z 131.06,A -85,B 0,C 180,E1 -660.163,E2 -660.163} C_VEL
LIN {X 0,Y 601.416,Z 131.068,A -85,B 0,C 180,E1 -662.715,E2 -662.715} C_VEL
LIN {X 0,Y 601.392,Z 131.077,A -85,B 0,C 180,E1 -665.112,E2 -665.112} C_VEL
LIN {X 0,Y 601.432,Z 131.066,A -85,B 0,C 180,E1 -667.419,E2 -667.419} C_VEL
LIN {X 0,Y 601.408,Z 131.065,A -85,B 0,C 180,E1 -669.995,E2 -669.995} C_VEL
LIN {X 0,Y 601.407,Z 131.07,A -85,B 0,C 180,E1 -672.67,E2 -672.67} C_VEL
LIN {X 0,Y 601.42,Z 131.065,A -85,B 0,C 180,E1 -675.482,E2 -675.482} C_VEL
LIN {X 0,Y 601.421,Z 131.069,A -85,B 0,C 180,E1 -678.407,E2 -678.407} C_VEL
LIN {X 0,Y 601.43,Z 131.069,A -85,B 0,C 180,E1 -680.875,E2 -680.875} C_VEL
LIN {X 0,Y 601.437,Z 131.062,A -85,B 0,C 180,E1 -683.734,E2 -683.734} C_VEL
LIN {X 0,Y 601.426,Z 131.07,A -85,B 0,C 180,E1 -686.687,E2 -686.687} C_VEL
LIN {X 0,Y 601.425,Z 131.065,A -85,B 0,C 180,E1 -689.059,E2 -689.059} C_VEL
LIN {X 0,Y 601.431,Z 131.062,A -85,B 0,C 180,E1 -691.374,E2 -691.374} C_VEL
LIN {X 0,Y 601.416,Z 131.071,A -85,B 0,C 180,E1 -694.131,E2 -694.131} C_VEL
LIN {X 0,Y 601.418,Z 131.068,A -85,B 0,C 180,E1 -696.59,E2 -696.59} C_VEL
LIN {X 0,Y 601.424,Z 131.064,A -85,B 0,C 180,E1 -699.478,E2 -699.478} C_VEL
LIN {X 0,Y 601.398,Z 131.073,A -85,B 0,C 180,E1 -702.312,E2 -702.312} C_VEL
LIN {X 0,Y 601.416,Z 131.068,A -85,B 0,C 180,E1 -704.409,E2 -704.409} C_VEL
LIN {X 0,Y 601.416,Z 131.065,A -85,B 0,C 180,E1 -707.172,E2 -707.172} C_VEL
LIN {X 0,Y 601.429,Z 131.072,A -85,B 0,C 180,E1 -709.905,E2 -709.905} C_VEL
LIN {X 0,Y 601.438,Z 131.062,A -85,B 0,C 180,E1 -712.615,E2 -712.615} C_VEL
LIN {X 0,Y 601.417,Z 131.068,A -85,B 0,C 180,E1 -715.308,E2 -715.308} C_VEL
LIN {X 0,Y 601.423,Z 131.067,A -85,B 0,C 180,E1 -717.991,E2 -717.991} C_VEL
LIN {X 0,Y 601.446,Z 131.059,A -85,B 0,C 180,E1 -720.67,E2 -720.67} C_VEL
LIN {X 0,Y 601.425,Z 131.07,A -85,B 0,C 180,E1 -723.35,E2 -723.35} C_VEL
LIN {X 0,Y 601.41,Z 131.067,A -85,B 0,C 180,E1 -726.037,E2 -726.037} C_VEL
LIN {X 0,Y 601.411,Z 131.065,A -85,B 0,C 180,E1 -728.738,E2 -728.738} C_VEL
LIN {X 0,Y 601.432,Z 131.07,A -85,B 0,C 180,E1 -731.459,E2 -731.459} C_VEL
LIN {X 0,Y 601.416,Z 131.064,A -85,B 0,C 180,E1 -734.206,E2 -734.206} C_VEL
LIN {X 0,Y 601.42,Z 131.071,A -85,B 0,C 180,E1 -736.987,E2 -736.987} C_VEL
LIN {X 0,Y 601.404,Z 131.066,A -85,B 0,C 180,E1 -739.81,E2 -739.81} C_VEL
LIN {X 0,Y 601.409,Z 131.07,A -85,B 0,C 180,E1 -742.683,E2 -742.683} C_VEL
LIN {X 0,Y 601.401,Z 131.075,A -85,B 0,C 180,E1 -744.879,E2 -744.879} C_VEL
LIN {X 0,Y 601.417,Z 131.067,A -85,B 0,C 180,E1 -747.364,E2 -747.364} C_VEL
LIN {X 0,Y 601.426,Z 131.064,A -85,B 0,C 180,E1 -750.164,E2 -750.164} C_VEL
LIN {X 0,Y 601.417,Z 131.074,A -85,B 0,C 180,E1 -752.716,E2 -752.716} C_VEL
LIN {X 0,Y 601.416,Z 131.068,A -85,B 0,C 180,E1 -755.116,E2 -755.116} C_VEL
LIN {X 0,Y 601.433,Z 131.063,A -85,B 0,C 180,E1 -757.42,E2 -757.42} C_VEL
LIN {X 0,Y 601.4,Z 131.068,A -85,B 0,C 180,E1 -759.996,E2 -759.996} C_VEL
LIN {X 0,Y 601.411,Z 131.072,A -85,B 0,C 180,E1 -762.671,E2 -762.671} C_VEL
LIN {X 0,Y 601.397,Z 131.066,A -85,B 0,C 180,E1 -765.48,E2 -765.48} C_VEL
LIN {X 0,Y 601.423,Z 131.072,A -85,B 0,C 180,E1 -768.407,E2 -768.407} C_VEL
LIN {X 0,Y 601.439,Z 131.063,A -85,B 0,C 180,E1 -770.876,E2 -770.876} C_VEL
LIN {X 0,Y 601.404,Z 131.066,A -85,B 0,C 180,E1 -773.418,E2 -773.418} C_VEL
LIN {X 0,Y 601.432,Z 131.071,A -85,B 0,C 180,E1 -776.065,E2 -776.065} C_VEL
LIN {X 0,Y 601.43,Z 131.063,A -85,B 0,C 180,E1 -779.059,E2 -779.059} C_VEL
LIN {X 0,Y 601.418,Z 131.066,A -85,B 0,C 180,E1 -781.373,E2 -781.373} C_VEL
LIN {X 0,Y 601.397,Z 131.073,A -85,B 0,C 180,E1 -783.636,E2 -783.636} C_VEL
LIN {X 0,Y 601.463,Z 131.238,A -85,B 0,C 180,E1 -785.703,E2 -785.703} C_VEL
LIN {X 0,Y 601.562,Z 140.545,A -85,B 0,C 180,E1 -787.362,E2 -787.362} C_VEL
LIN {X 0,Y 601.529,Z 155.846,A -85,B 0,C 180,E1 -790.017,E2 -790.017} C_VEL
LIN {X 0,Y 601.468,Z 172.403,A -85,B 0,C 180,E1 -792.84,E2 -792.84} C_VEL
LIN {X 0,Y 601.456,Z 187.924,A -85,B 0,C 180,E1 -795.45,E2 -795.45} C_VEL
LIN {X 0,Y 601.451,Z 196.24,A -85,B 0,C 180,E1 -796.808,E2 -796.808} C_VEL
LIN {X 0,Y 601.633,Z 198.731,A -85,B 0,C 180,E1 -796.876,E2 -796.876} C_VEL
LIN {X 0,Y 601.617,Z 302.883,A -85,B 0,C 180,E1 -798.14,E2 -798.14} C_VEL
LIN {X 0,Y 601.591,Z 316.242,A -85,B 0,C 180,E1 -798.438,E2 -798.438} C_VEL
LIN {X 0,Y 601.548,Z 328.668,A -85,B 0,C 180,E1 -798.854,E2 -798.854} C_VEL
LIN {X 0,Y 601.52,Z 340.601,A -85,B 0,C 180,E1 -799.396,E2 -799.396} C_VEL
LIN {X 0,Y 601.481,Z 352.202,A -85,B 0,C 180,E1 -800.076,E2 -800.076} C_VEL
LIN {X 0,Y 601.438,Z 363.645,A -85,B 0,C 180,E1 -800.924,E2 -800.924} C_VEL
LIN {X 0,Y 601.411,Z 372.775,A -85,B 0,C 180,E1 -801.77,E2 -801.77} C_VEL
LIN {X 0,Y 601.388,Z 381.681,A -85,B 0,C 180,E1 -802.783,E2 -802.783} C_VEL
LIN {X 0,Y 601.375,Z 388.773,A -85,B 0,C 180,E1 -803.782,E2 -803.782} C_VEL
LIN {X 0,Y 601.345,Z 395.365,A -85,B 0,C 180,E1 -804.971,E2 -804.971} C_VEL
LIN {X 0,Y 601.347,Z 399.671,A -85,B 0,C 180,E1 -805.979,E2 -805.979} C_VEL
LIN {X 0,Y 601.344,Z 401.96,A -85,B 0,C 180,E1 -806.65,E2 -806.65} C_VEL
LIN {X 0,Y 601.325,Z 403.803,A -85,B 0,C 180,E1 -807.32,E2 -807.32} C_VEL
LIN {X 0,Y 601.343,Z 405.198,A -85,B 0,C 180,E1 -807.991,E2 -807.991} C_VEL
LIN {X 0,Y 601.347,Z 406.186,A -85,B 0,C 180,E1 -808.661,E2 -808.661} C_VEL
LIN {X 0,Y 601.335,Z 406.988,A -85,B 0,C 180,E1 -810,E2 -810} C_VEL
LIN {X 0,Y 601.347,Z 406.186,A -85,B 0,C 180,E1 -811.339,E2 -811.339} C_VEL
LIN {X 0,Y 601.343,Z 405.198,A -85,B 0,C 180,E1 -812.009,E2 -812.009} C_VEL
LIN {X 0,Y 601.325,Z 403.803,A -85,B 0,C 180,E1 -812.68,E2 -812.68} C_VEL
LIN {X 0,Y 601.368,Z 400.893,A -85,B 0,C 180,E1 -813.685,E2 -813.685} C_VEL
LIN {X 0,Y 601.336,Z 396.947,A -85,B 0,C 180,E1 -814.693,E2 -814.693} C_VEL
LIN {X 0,Y 601.374,Z 391.854,A -85,B 0,C 180,E1 -815.701,E2 -815.701} C_VEL
LIN {X 0,Y 601.382,Z 385.468,A -85,B 0,C 180,E1 -816.711,E2 -816.711} C_VEL
LIN {X 0,Y 601.396,Z 377.484,A -85,B 0,C 180,E1 -817.723,E2 -817.723} C_VEL
LIN {X 0,Y 601.423,Z 369.343,A -85,B 0,C 180,E1 -818.568,E2 -818.568} C_VEL
LIN {X 0,Y 601.454,Z 359.38,A -85,B 0,C 180,E1 -819.415,E2 -819.415} C_VEL
LIN {X 0,Y 601.478,Z 349.565,A -85,B 0,C 180,E1 -820.094,E2 -820.094} C_VEL
LIN {X 0,Y 601.53,Z 338.932,A -85,B 0,C 180,E1 -820.689,E2 -820.689} C_VEL
LIN {X 0,Y 601.572,Z 325.571,A -85,B 0,C 180,E1 -821.263,E2 -821.263} C_VEL
LIN {X 0,Y 601.593,Z 313.029,A -85,B 0,C 180,E1 -821.647,E2 -821.647} C_VEL
LIN {X 0,Y 601.634,Z 300.117,A -85,B 0,C 180,E1 -821.903,E2 -821.903} C_VEL
LIN {X 0,Y 601.526,Z 197.221,A -85,B 0,C 180,E1 -823.148,E2 -823.148} C_VEL
LIN {X 0,Y 601.415,Z 196.028,A -85,B 0,C 180,E1 -823.215,E2 -823.215} C_VEL
LIN {X 0,Y 601.486,Z 179.646,A -85,B 0,C 180,E1 -825.937,E2 -825.937} C_VEL
LIN {X 0,Y 601.525,Z 162.465,A -85,B 0,C 180,E1 -828.848,E2 -828.848} C_VEL
LIN {X 0,Y 601.557,Z 145.498,A -85,B 0,C 180,E1 -831.773,E2 -831.773} C_VEL
LIN {X 0,Y 601.601,Z 132.046,A -85,B 0,C 180,E1 -834.134,E2 -834.134} C_VEL
LIN {X 0,Y 601.423,Z 131.109,A -85,B 0,C 180,E1 -834.383,E2 -834.383} C_VEL
LIN {X 0,Y 601.449,Z 131.061,A -85,B 0,C 180,E1 -837.111,E2 -837.111} C_VEL
LIN {X 0,Y 601.43,Z 131.07,A -85,B 0,C 180,E1 -840.164,E2 -840.164} C_VEL
LIN {X 0,Y 601.412,Z 131.065,A -85,B 0,C 180,E1 -842.713,E2 -842.713} C_VEL
LIN {X 0,Y 601.396,Z 131.067,A -85,B 0,C 180,E1 -845.111,E2 -845.111} C_VEL
LIN {X 0,Y 601.435,Z 131.066,A -85,B 0,C 180,E1 -847.419,E2 -847.419} C_VEL
LIN {X 0,Y 601.413,Z 131.069,A -85,B 0,C 180,E1 -849.994,E2 -849.994} C_VEL
LIN {X 0,Y 601.408,Z 131.065,A -85,B 0,C 180,E1 -852.67,E2 -852.67} C_VEL
LIN {X 0,Y 601.426,Z 131.072,A -85,B 0,C 180,E1 -855.482,E2 -855.482} C_VEL
LIN {X 0,Y 601.421,Z 131.064,A -85,B 0,C 180,E1 -858.407,E2 -858.407} C_VEL
LIN {X 0,Y 601.427,Z 131.071,A -85,B 0,C 180,E1 -861.529,E2 -861.529} C_VEL
LIN {X 0,Y 601.388,Z 131.068,A -85,B 0,C 180,E1 -864.245,E2 -864.245} C_VEL
LIN {X 0,Y 601.426,Z 131.064,A -85,B 0,C 180,E1 -866.686,E2 -866.686} C_VEL
LIN {X 0,Y 601.429,Z 131.071,A -85,B 0,C 180,E1 -869.058,E2 -869.058} C_VEL
LIN {X 0,Y 601.426,Z 131.069,A -85,B 0,C 180,E1 -871.373,E2 -871.373} C_VEL
LIN {X 0,Y 601.4,Z 131.068,A -85,B 0,C 180,E1 -873.636,E2 -873.636} C_VEL
LIN {X 0,Y 601.417,Z 131.068,A -85,B 0,C 180,E1 -876.589,E2 -876.589} C_VEL
LIN {X 0,Y 601.422,Z 131.065,A -85,B 0,C 180,E1 -879.478,E2 -879.478} C_VEL
LIN {X 0,Y 601.4,Z 131.067,A -85,B 0,C 180,E1 -882.311,E2 -882.311} C_VEL
LIN {X 0,Y 601.425,Z 131.068,A -85,B 0,C 180,E1 -885.103,E2 -885.103} C_VEL
LIN {X 0,Y 601.414,Z 131.064,A -85,B 0,C 180,E1 -887.857,E2 -887.857} C_VEL
LIN {X 0,Y 601.416,Z 131.073,A -85,B 0,C 180,E1 -890.584,E2 -890.584} C_VEL
LIN {X 0,Y 601.452,Z 131.06,A -85,B 0,C 180,E1 -893.323,E2 -893.323} C_VEL
LIN {X 0,Y 601.405,Z 131.068,A -85,B 0,C 180,E1 -895.979,E2 -895.979} C_VEL
LIN {X 0,Y 601.417,Z 131.069,A -85,B 0,C 180,E1 -898.66,E2 -898.66} C_VEL
LIN {X 0,Y 601.424,Z 131.062,A -85,B 0,C 180,E1 -901.339,E2 -901.339} C_VEL
LIN {X 0,Y 601.404,Z 131.071,A -85,B 0,C 180,E1 -904.02,E2 -904.02} C_VEL
LIN {X 0,Y 601.422,Z 131.066,A -85,B 0,C 180,E1 -906.71,E2 -906.71} C_VEL
LIN {X 0,Y 601.42,Z 131.064,A -85,B 0,C 180,E1 -909.449,E2 -909.449} C_VEL
LIN {X 0,Y 601.415,Z 131.073,A -85,B 0,C 180,E1 -912.142,E2 -912.142} C_VEL
LIN {X 0,Y 601.405,Z 131.07,A -85,B 0,C 180,E1 -912.368,E2 -912.368} C_VEL
LIN {X 0,Y 600.739,Z 131.151,A -85,B 0,C 180,E1 -912.928,E2 -912.928} C_VEL
LIN {X 0,Y 597.889,Z 131.511,A -85,B 0,C 180,E1 -913.836,E2 -913.836} C_VEL
LIN {X 0,Y 595.48,Z 131.806,A -85,B 0,C 180,E1 -914.566,E2 -914.566} C_VEL
LIN {X 0,Y 594.444,Z 131.933,A -85,B 0,C 180,E1 -915.129,E2 -915.129} C_VEL
LIN {X 0,Y 594.359,Z 131.945,A -85,B 0,C 180,E1 -915.32,E2 -915.32} C_VEL
LIN {X 0,Y 594.379,Z 131.95,A -85,B 0,C 180,E1 -917.904,E2 -917.904} C_VEL
LIN {X 0,Y 594.374,Z 131.941,A -85,B 0,C 180,E1 -920.916,E2 -920.916} C_VEL
LIN {X 0,Y 594.386,Z 131.95,A -85,B 0,C 180,E1 -923.704,E2 -923.704} C_VEL
LIN {X 0,Y 594.381,Z 131.939,A -85,B 0,C 180,E1 -926.699,E2 -926.699} C_VEL
LIN {X 0,Y 594.377,Z 131.942,A -85,B 0,C 180,E1 -928.998,E2 -928.998} C_VEL
LIN {X 0,Y 594.387,Z 131.948,A -85,B 0,C 180,E1 -931.645,E2 -931.645} C_VEL
LIN {X 0,Y 594.391,Z 131.938,A -85,B 0,C 180,E1 -934.579,E2 -934.579} C_VEL
LIN {X 0,Y 594.381,Z 131.946,A -85,B 0,C 180,E1 -937.086,E2 -937.086} C_VEL
LIN {X 0,Y 594.369,Z 131.945,A -85,B 0,C 180,E1 -939.774,E2 -939.774} C_VEL
LIN {X 0,Y 594.384,Z 131.94,A -85,B 0,C 180,E1 -942.373,E2 -942.373} C_VEL
LIN {X 0,Y 594.359,Z 131.953,A -85,B 0,C 180,E1 -945.191,E2 -945.191} C_VEL
LIN {X 0,Y 594.379,Z 131.938,A -85,B 0,C 180,E1 -948.151,E2 -948.151} C_VEL
LIN {X 0,Y 594.385,Z 131.948,A -85,B 0,C 180,E1 -951.196,E2 -951.196} C_VEL
LIN {X 0,Y 594.392,Z 131.939,A -85,B 0,C 180,E1 -953.759,E2 -953.759} C_VEL
LIN {X 0,Y 594.376,Z 131.941,A -85,B 0,C 180,E1 -956.239,E2 -956.239} C_VEL
LIN {X 0,Y 594.388,Z 131.947,A -85,B 0,C 180,E1 -958.651,E2 -958.651} C_VEL
LIN {X 0,Y 594.379,Z 131.946,A -85,B 0,C 180,E1 -961.042,E2 -961.042} C_VEL
LIN {X 0,Y 594.382,Z 131.942,A -85,B 0,C 180,E1 -963.977,E2 -963.977} C_VEL
LIN {X 0,Y 594.387,Z 131.945,A -85,B 0,C 180,E1 -966.296,E2 -966.296} C_VEL
LIN {X 0,Y 594.403,Z 131.939,A -85,B 0,C 180,E1 -969.225,E2 -969.225} C_VEL
LIN {X 0,Y 594.351,Z 131.949,A -85,B 0,C 180,E1 -972.095,E2 -972.095} C_VEL
LIN {X 0,Y 594.364,Z 131.95,A -85,B 0,C 180,E1 -974.219,E2 -974.219} C_VEL
LIN {X 0,Y 594.365,Z 131.944,A -85,B 0,C 180,E1 -977.017,E2 -977.017} C_VEL
LIN {X 0,Y 594.395,Z 131.942,A -85,B 0,C 180,E1 -979.784,E2 -979.784} C_VEL
LIN {X 0,Y 594.39,Z 131.945,A -85,B 0,C 180,E1 -982.527,E2 -982.527} C_VEL
LIN {X 0,Y 594.389,Z 131.94,A -85,B 0,C 180,E1 -985.252,E2 -985.252} C_VEL
LIN {X 0,Y 594.404,Z 131.947,A -85,B 0,C 180,E1 -987.967,E2 -987.967} C_VEL
LIN {X 0,Y 594.418,Z 131.937,A -85,B 0,C 180,E1 -990.677,E2 -990.677} C_VEL
LIN {X 0,Y 594.377,Z 131.944,A -85,B 0,C 180,E1 -993.389,E2 -993.389} C_VEL
LIN {X 0,Y 594.375,Z 131.947,A -85,B 0,C 180,E1 -996.109,E2 -996.109} C_VEL
LIN {X 0,Y 594.395,Z 131.939,A -85,B 0,C 180,E1 -998.842,E2 -998.842} C_VEL
LIN {X 0,Y 594.391,Z 131.948,A -85,B 0,C 180,E1 -1001.596,E2 -1001.596} C_VEL
LIN {X 0,Y 594.387,Z 131.941,A -85,B 0,C 180,E1 -1004.377,E2 -1004.377} C_VEL
LIN {X 0,Y 594.387,Z 131.945,A -85,B 0,C 180,E1 -1007.193,E2 -1007.193} C_VEL
LIN {X 0,Y 594.373,Z 131.944,A -85,B 0,C 180,E1 -1010.054,E2 -1010.054} C_VEL
LIN {X 0,Y 594.361,Z 131.947,A -85,B 0,C 180,E1 -1012.967,E2 -1012.967} C_VEL
LIN {X 0,Y 594.372,Z 131.95,A -85,B 0,C 180,E1 -1015.193,E2 -1015.193} C_VEL
LIN {X 0,Y 594.381,Z 131.946,A -85,B 0,C 180,E1 -1017.527,E2 -1017.527} C_VEL
LIN {X 0,Y 594.392,Z 131.94,A -85,B 0,C 180,E1 -1020.559,E2 -1020.559} C_VEL
LIN {X 0,Y 594.374,Z 131.949,A -85,B 0,C 180,E1 -1022.95,E2 -1022.95} C_VEL
LIN {X 0,Y 594.351,Z 131.948,A -85,B 0,C 180,E1 -1025.408,E2 -1025.408} C_VEL
LIN {X 0,Y 594.385,Z 131.94,A -85,B 0,C 180,E1 -1027.94,E2 -1027.94} C_VEL
LIN {X 0,Y 594.376,Z 131.949,A -85,B 0,C 180,E1 -1030.823,E2 -1030.823} C_VEL
LIN {X 0,Y 594.362,Z 131.945,A -85,B 0,C 180,E1 -1033.299,E2 -1033.299} C_VEL
LIN {X 0,Y 594.377,Z 131.943,A -85,B 0,C 180,E1 -1036.159,E2 -1036.159} C_VEL
LIN {X 0,Y 594.378,Z 131.948,A -85,B 0,C 180,E1 -1038.537,E2 -1038.537} C_VEL
LIN {X 0,Y 594.382,Z 131.942,A -85,B 0,C 180,E1 -1041.295,E2 -1041.295} C_VEL
LIN {X 0,Y 594.39,Z 131.94,A -85,B 0,C 180,E1 -1043.759,E2 -1043.759} C_VEL
LIN {X 0,Y 594.379,Z 131.945,A -85,B 0,C 180,E1 -1046.239,E2 -1046.239} C_VEL
LIN {X 0,Y 594.385,Z 131.947,A -85,B 0,C 180,E1 -1048.651,E2 -1048.651} C_VEL
LIN {X 0,Y 594.38,Z 131.941,A -85,B 0,C 180,E1 -1051.042,E2 -1051.042} C_VEL
LIN {X 0,Y 594.389,Z 131.943,A -85,B 0,C 180,E1 -1053.976,E2 -1053.976} C_VEL
LIN {X 0,Y 594.386,Z 131.95,A -85,B 0,C 180,E1 -1056.296,E2 -1056.296} C_VEL
LIN {X 0,Y 594.398,Z 131.938,A -85,B 0,C 180,E1 -1059.225,E2 -1059.225} C_VEL
LIN {X 0,Y 594.378,Z 131.95,A -85,B 0,C 180,E1 -1062.096,E2 -1062.096} C_VEL
LIN {X 0,Y 594.368,Z 131.949,A -85,B 0,C 180,E1 -1064.22,E2 -1064.22} C_VEL
LIN {X 0,Y 594.364,Z 131.942,A -85,B 0,C 180,E1 -1067.017,E2 -1067.017} C_VEL
LIN {X 0,Y 594.388,Z 131.947,A -85,B 0,C 180,E1 -1069.784,E2 -1069.784} C_VEL
LIN {X 0,Y 594.391,Z 131.94,A -85,B 0,C 180,E1 -1072.527,E2 -1072.527} C_VEL
LIN {X 0,Y 594.387,Z 131.943,A -85,B 0,C 180,E1 -1075.253,E2 -1075.253} C_VEL
LIN {X 0,Y 594.393,Z 131.943,A -85,B 0,C 180,E1 -1077.968,E2 -1077.968} C_VEL
LIN {X 0,Y 594.417,Z 131.934,A -85,B 0,C 180,E1 -1080.678,E2 -1080.678} C_VEL
LIN {X 0,Y 594.377,Z 131.948,A -85,B 0,C 180,E1 -1083.39,E2 -1083.39} C_VEL
LIN {X 0,Y 594.366,Z 131.943,A -85,B 0,C 180,E1 -1086.109,E2 -1086.109} C_VEL
LIN {X 0,Y 594.378,Z 131.942,A -85,B 0,C 180,E1 -1088.843,E2 -1088.843} C_VEL
LIN {X 0,Y 594.391,Z 131.944,A -85,B 0,C 180,E1 -1091.596,E2 -1091.596} C_VEL
LIN {X 0,Y 594.386,Z 131.94,A -85,B 0,C 180,E1 -1094.377,E2 -1094.377} C_VEL
LIN {X 0,Y 594.383,Z 131.949,A -85,B 0,C 180,E1 -1097.194,E2 -1097.194} C_VEL
LIN {X 0,Y 594.371,Z 131.941,A -85,B 0,C 180,E1 -1100.054,E2 -1100.054} C_VEL
LIN {X 0,Y 594.362,Z 131.953,A -85,B 0,C 180,E1 -1102.968,E2 -1102.968} C_VEL
LIN {X 0,Y 594.377,Z 131.946,A -85,B 0,C 180,E1 -1105.193,E2 -1105.193} C_VEL
LIN {X 0,Y 594.383,Z 131.941,A -85,B 0,C 180,E1 -1107.527,E2 -1107.527} C_VEL
LIN {X 0,Y 594.386,Z 131.943,A -85,B 0,C 180,E1 -1110.329,E2 -1110.329} C_VEL
LIN {X 0,Y 594.376,Z 131.947,A -85,B 0,C 180,E1 -1112.951,E2 -1112.951} C_VEL
LIN {X 0,Y 594.356,Z 131.944,A -85,B 0,C 180,E1 -1115.409,E2 -1115.409} C_VEL
LIN {X 0,Y 594.38,Z 131.942,A -85,B 0,C 180,E1 -1117.942,E2 -1117.942} C_VEL
LIN {X 0,Y 594.376,Z 131.947,A -85,B 0,C 180,E1 -1120.823,E2 -1120.823} C_VEL
LIN {X 0,Y 594.366,Z 131.943,A -85,B 0,C 180,E1 -1123.3,E2 -1123.3} C_VEL
LIN {X 0,Y 594.359,Z 131.949,A -85,B 0,C 180,E1 -1126.162,E2 -1126.162} C_VEL
LIN {X 0,Y 594.38,Z 131.946,A -85,B 0,C 180,E1 -1128.537,E2 -1128.537} C_VEL
LIN {X 0,Y 594.388,Z 131.94,A -85,B 0,C 180,E1 -1131.296,E2 -1131.296} C_VEL
LIN {X 0,Y 594.352,Z 131.947,A -85,B 0,C 180,E1 -1133.756,E2 -1133.756} C_VEL
LIN {X 0,Y 594.379,Z 131.949,A -85,B 0,C 180,E1 -1136.239,E2 -1136.239} C_VEL
LIN {X 0,Y 594.391,Z 131.942,A -85,B 0,C 180,E1 -1138.651,E2 -1138.651} C_VEL
LIN {X 0,Y 594.379,Z 131.942,A -85,B 0,C 180,E1 -1141.044,E2 -1141.044} C_VEL
LIN {X 0,Y 594.382,Z 131.943,A -85,B 0,C 180,E1 -1143.301,E2 -1143.301} C_VEL
LIN {X 0,Y 594.396,Z 132.118,A -85,B 0,C 180,E1 -1145.565,E2 -1145.565} C_VEL
LIN {X 0,Y 594.665,Z 136.157,A -85,B 0,C 180,E1 -1146.308,E2 -1146.308} C_VEL
LIN {X 0,Y 594.544,Z 152.742,A -85,B 0,C 180,E1 -1149.23,E2 -1149.23} C_VEL
LIN {X 0,Y 594.464,Z 167.229,A -85,B 0,C 180,E1 -1151.742,E2 -1151.742} C_VEL
LIN {X 0,Y 594.447,Z 183.785,A -85,B 0,C 180,E1 -1154.573,E2 -1154.573} C_VEL
LIN {X 0,Y 594.41,Z 196.235,A -85,B 0,C 180,E1 -1156.648,E2 -1156.648} C_VEL
LIN {X 0,Y 594.726,Z 198.731,A -85,B 0,C 180,E1 -1156.721,E2 -1156.721} C_VEL
LIN {X 0,Y 594.669,Z 302.816,A -85,B 0,C 180,E1 -1157.999,E2 -1157.999} C_VEL
LIN {X 0,Y 594.626,Z 315.494,A -85,B 0,C 180,E1 -1158.279,E2 -1158.279} C_VEL
LIN {X 0,Y 594.593,Z 329.329,A -85,B 0,C 180,E1 -1158.748,E2 -1158.748} C_VEL
LIN {X 0,Y 594.537,Z 340.58,A -85,B 0,C 180,E1 -1159.27,E2 -1159.27} C_VEL
LIN {X 0,Y 594.452,Z 350.894,A -85,B 0,C 180,E1 -1159.871,E2 -1159.871} C_VEL
LIN {X 0,Y 594.406,Z 361.545,A -85,B 0,C 180,E1 -1160.644,E2 -1160.644} C_VEL
LIN {X 0,Y 594.383,Z 371.121,A -85,B 0,C 180,E1 -1161.501,E2 -1161.501} C_VEL
LIN {X 0,Y 594.347,Z 378.944,A -85,B 0,C 180,E1 -1162.355,E2 -1162.355} C_VEL
LIN {X 0,Y 594.303,Z 386.69,A -85,B 0,C 180,E1 -1163.391,E2 -1163.391} C_VEL
LIN {X 0,Y 594.289,Z 393.682,A -85,B 0,C 180,E1 -1164.571,E2 -1164.571} C_VEL
LIN {X 0,Y 594.27,Z 398.377,A -85,B 0,C 180,E1 -1165.591,E2 -1165.591} C_VEL
LIN {X 0,Y 594.267,Z 401.963,A -85,B 0,C 180,E1 -1166.61,E2 -1166.61} C_VEL
LIN {X 0,Y 594.225,Z 403.797,A -85,B 0,C 180,E1 -1167.288,E2 -1167.288} C_VEL
LIN {X 0,Y 594.247,Z 406.188,A -85,B 0,C 180,E1 -1168.645,E2 -1168.645} C_VEL
LIN {X 0,Y 594.239,Z 406.782,A -85,B 0,C 180,E1 -1169.322,E2 -1169.322} C_VEL
LIN {X 0,Y 594.236,Z 406.979,A -85,B 0,C 180,E1 -1170,E2 -1170} C_VEL
LIN {X 0,Y 594.239,Z 406.782,A -85,B 0,C 180,E1 -1170.678,E2 -1170.678} C_VEL
LIN {X 0,Y 594.247,Z 406.188,A -85,B 0,C 180,E1 -1171.355,E2 -1171.355} C_VEL
LIN {X 0,Y 594.225,Z 403.797,A -85,B 0,C 180,E1 -1172.712,E2 -1172.712} C_VEL
LIN {X 0,Y 594.289,Z 400.886,A -85,B 0,C 180,E1 -1173.729,E2 -1173.729} C_VEL
LIN {X 0,Y 594.241,Z 396.938,A -85,B 0,C 180,E1 -1174.749,E2 -1174.749} C_VEL
LIN {X 0,Y 594.3,Z 391.843,A -85,B 0,C 180,E1 -1175.769,E2 -1175.769} C_VEL
LIN {X 0,Y 594.316,Z 385.459,A -85,B 0,C 180,E1 -1176.791,E2 -1176.791} C_VEL
LIN {X 0,Y 594.346,Z 377.488,A -85,B 0,C 180,E1 -1177.815,E2 -1177.815} C_VEL
LIN {X 0,Y 594.378,Z 369.347,A -85,B 0,C 180,E1 -1178.671,E2 -1178.671} C_VEL
LIN {X 0,Y 594.417,Z 359.364,A -85,B 0,C 180,E1 -1179.528,E2 -1179.528} C_VEL
LIN {X 0,Y 594.467,Z 349.546,A -85,B 0,C 180,E1 -1180.214,E2 -1180.214} C_VEL
LIN {X 0,Y 594.55,Z 338.937,A -85,B 0,C 180,E1 -1180.816,E2 -1180.816} C_VEL
LIN {X 0,Y 594.598,Z 326.056,A -85,B 0,C 180,E1 -1181.379,E2 -1181.379} C_VEL
LIN {X 0,Y 594.654,Z 313.863,A -85,B 0,C 180,E1 -1181.763,E2 -1181.763} C_VEL
LIN {X 0,Y 594.675,Z 301.485,A -85,B 0,C 180,E1 -1182.022,E2 -1182.022} C_VEL
LIN {X 0,Y 594.573,Z 197.643,A -85,B 0,C 180,E1 -1183.296,E2 -1183.296} C_VEL
LIN {X 0,Y 594.399,Z 196.025,A -85,B 0,C 180,E1 -1183.374,E2 -1183.374} C_VEL
LIN {X 0,Y 594.448,Z 179.646,A -85,B 0,C 180,E1 -1186.131,E2 -1186.131} C_VEL
LIN {X 0,Y 594.53,Z 163.093,A -85,B 0,C 180,E1 -1188.97,E2 -1188.97} C_VEL
LIN {X 0,Y 594.587,Z 147.568,A -85,B 0,C 180,E1 -1191.677,E2 -1191.677} C_VEL
LIN {X 0,Y 594.67,Z 134.097,A -85,B 0,C 180,E1 -1194.057,E2 -1194.057} C_VEL
LIN {X 0,Y 594.387,Z 131.999,A -85,B 0,C 180,E1 -1194.492,E2 -1194.492} C_VEL
LIN {X 0,Y 594.382,Z 131.943,A -85,B 0,C 180,E1 -1196.699,E2 -1196.699} C_VEL
LIN {X 0,Y 594.377,Z 131.942,A -85,B 0,C 180,E1 -1198.998,E2 -1198.998} C_VEL
LIN {X 0,Y 594.391,Z 131.945,A -85,B 0,C 180,E1 -1201.644,E2 -1201.644} C_VEL
LIN {X 0,Y 594.379,Z 131.941,A -85,B 0,C 180,E1 -1204.58,E2 -1204.58} C_VEL
LIN {X 0,Y 594.389,Z 131.947,A -85,B 0,C 180,E1 -1207.608,E2 -1207.608} C_VEL
LIN {X 0,Y 594.378,Z 131.949,A -85,B 0,C 180,E1 -1209.774,E2 -1209.774} C_VEL
LIN {X 0,Y 594.364,Z 131.943,A -85,B 0,C 180,E1 -1212.375,E2 -1212.375} C_VEL
LIN {X 0,Y 594.355,Z 131.948,A -85,B 0,C 180,E1 -1215.192,E2 -1215.192} C_VEL
LIN {X 0,Y 594.377,Z 131.942,A -85,B 0,C 180,E1 -1218.152,E2 -1218.152} C_VEL
LIN {X 0,Y 594.376,Z 131.947,A -85,B 0,C 180,E1 -1221.194,E2 -1221.194} C_VEL
LIN {X 0,Y 594.35,Z 131.948,A -85,B 0,C 180,E1 -1223.755,E2 -1223.755} C_VEL
LIN {X 0,Y 594.379,Z 131.94,A -85,B 0,C 180,E1 -1226.238,E2 -1226.238} C_VEL
LIN {X 0,Y 594.389,Z 131.942,A -85,B 0,C 180,E1 -1228.65,E2 -1228.65} C_VEL
LIN {X 0,Y 594.381,Z 131.949,A -85,B 0,C 180,E1 -1231.042,E2 -1231.042} C_VEL
LIN {X 0,Y 594.387,Z 131.939,A -85,B 0,C 180,E1 -1233.976,E2 -1233.976} C_VEL
LIN {X 0,Y 594.386,Z 131.941,A -85,B 0,C 180,E1 -1236.295,E2 -1236.295} C_VEL
LIN {X 0,Y 594.395,Z 131.943,A -85,B 0,C 180,E1 -1239.224,E2 -1239.224} C_VEL
LIN {X 0,Y 594.378,Z 131.94,A -85,B 0,C 180,E1 -1242.095,E2 -1242.095} C_VEL
LIN {X 0,Y 594.368,Z 131.944,A -85,B 0,C 180,E1 -1244.219,E2 -1244.219} C_VEL
LIN {X 0,Y 594.366,Z 131.947,A -85,B 0,C 180,E1 -1247.017,E2 -1247.017} C_VEL
LIN {X 0,Y 594.388,Z 131.938,A -85,B 0,C 180,E1 -1249.784,E2 -1249.784} C_VEL
LIN {X 0,Y 594.39,Z 131.948,A -85,B 0,C 180,E1 -1252.526,E2 -1252.526} C_VEL
LIN {X 0,Y 594.389,Z 131.94,A -85,B 0,C 180,E1 -1255.252,E2 -1255.252} C_VEL
LIN {X 0,Y 594.393,Z 131.942,A -85,B 0,C 180,E1 -1257.967,E2 -1257.967} C_VEL
LIN {X 0,Y 594.416,Z 131.94,A -85,B 0,C 180,E1 -1260.677,E2 -1260.677} C_VEL
LIN {X 0,Y 594.38,Z 131.94,A -85,B 0,C 180,E1 -1263.389,E2 -1263.389} C_VEL
LIN {X 0,Y 594.362,Z 131.951,A -85,B 0,C 180,E1 -1266.109,E2 -1266.109} C_VEL
LIN {X 0,Y 594.379,Z 131.94,A -85,B 0,C 180,E1 -1268.842,E2 -1268.842} C_VEL
LIN {X 0,Y 594.393,Z 131.941,A -85,B 0,C 180,E1 -1271.595,E2 -1271.595} C_VEL
LIN {X 0,Y 594.385,Z 131.944,A -85,B 0,C 180,E1 -1274.377,E2 -1274.377} C_VEL
LIN {X 0,Y 594.359,Z 131.945,A -85,B 0,C 180,E1 -1275.32,E2 -1275.32} C_VEL
LIN {X 0,Y 593.691,Z 132.036,A -85,B 0,C 180,E1 -1275.886,E2 -1275.886} C_VEL
LIN {X 0,Y 590.839,Z 132.391,A -85,B 0,C 180,E1 -1276.804,E2 -1276.804} C_VEL
LIN {X 0,Y 588.433,Z 132.69,A -85,B 0,C 180,E1 -1277.543,E2 -1277.543} C_VEL
LIN {X 0,Y 587.403,Z 132.814,A -85,B 0,C 180,E1 -1278.113,E2 -1278.113} C_VEL
LIN {X 0,Y 587.321,Z 132.821,A -85,B 0,C 180,E1 -1278.306,E2 -1278.306} C_VEL
LIN {X 0,Y 587.325,Z 132.819,A -85,B 0,C 180,E1 -1281.037,E2 -1281.037} C_VEL
LIN {X 0,Y 587.318,Z 132.823,A -85,B 0,C 180,E1 -1283.258,E2 -1283.258} C_VEL
LIN {X 0,Y 587.335,Z 132.825,A -85,B 0,C 180,E1 -1285.516,E2 -1285.516} C_VEL
LIN {X 0,Y 587.343,Z 132.824,A -85,B 0,C 180,E1 -1287.817,E2 -1287.817} C_VEL
LIN {X 0,Y 587.336,Z 132.818,A -85,B 0,C 180,E1 -1290.511,E2 -1290.511} C_VEL
LIN {X 0,Y 587.336,Z 132.822,A -85,B 0,C 180,E1 -1293.112,E2 -1293.112} C_VEL
LIN {X 0,Y 587.351,Z 132.819,A -85,B 0,C 180,E1 -1295.895,E2 -1295.895} C_VEL
LIN {X 0,Y 587.327,Z 132.82,A -85,B 0,C 180,E1 -1298.479,E2 -1298.479} C_VEL
LIN {X 0,Y 587.332,Z 132.825,A -85,B 0,C 180,E1 -1301.157,E2 -1301.157} C_VEL
LIN {X 0,Y 587.329,Z 132.819,A -85,B 0,C 180,E1 -1304.114,E2 -1304.114} C_VEL
LIN {X 0,Y 587.31,Z 132.828,A -85,B 0,C 180,E1 -1306.994,E2 -1306.994} C_VEL
LIN {X 0,Y 587.315,Z 132.821,A -85,B 0,C 180,E1 -1309.746,E2 -1309.746} C_VEL
LIN {X 0,Y 587.342,Z 132.819,A -85,B 0,C 180,E1 -1312.393,E2 -1312.393} C_VEL
LIN {X 0,Y 587.344,Z 132.825,A -85,B 0,C 180,E1 -1314.946,E2 -1314.946} C_VEL
LIN {X 0,Y 587.335,Z 132.821,A -85,B 0,C 180,E1 -1317.421,E2 -1317.421} C_VEL
LIN {X 0,Y 587.343,Z 132.817,A -85,B 0,C 180,E1 -1319.831,E2 -1319.831} C_VEL
LIN {X 0,Y 587.348,Z 132.82,A -85,B 0,C 180,E1 -1322.307,E2 -1322.307} C_VEL
LIN {X 0,Y 587.331,Z 132.826,A -85,B 0,C 180,E1 -1324.484,E2 -1324.484} C_VEL
LIN {X 0,Y 587.315,Z 132.824,A -85,B 0,C 180,E1 -1327.131,E2 -1327.131} C_VEL
LIN {X 0,Y 587.329,Z 132.82,A -85,B 0,C 180,E1 -1329.695,E2 -1329.695} C_VEL
LIN {X 0,Y 587.347,Z 132.825,A -85,B 0,C 180,E1 -1332.594,E2 -1332.594} C_VEL
LIN {X 0,Y 587.362,Z 132.817,A -85,B 0,C 180,E1 -1335.74,E2 -1335.74} C_VEL
LIN {X 0,Y 587.345,Z 132.82,A -85,B 0,C 180,E1 -1338.866,E2 -1338.866} C_VEL
LIN {X 0,Y 587.368,Z 132.818,A -85,B 0,C 180,E1 -1341.745,E2 -1341.745} C_VEL
LIN {X 0,Y 587.356,Z 132.821,A -85,B 0,C 180,E1 -1344.507,E2 -1344.507} C_VEL
LIN {X 0,Y 587.37,Z 132.815,A -85,B 0,C 180,E1 -1347.257,E2 -1347.257} C_VEL
LIN {X 0,Y 587.382,Z 132.823,A -85,B 0,C 180,E1 -1350,E2 -1350} C_VEL
LIN {X 0,Y 587.37,Z 132.815,A -85,B 0,C 180,E1 -1352.743,E2 -1352.743} C_VEL
LIN {X 0,Y 587.356,Z 132.821,A -85,B 0,C 180,E1 -1355.493,E2 -1355.493} C_VEL
LIN {X 0,Y 587.368,Z 132.818,A -85,B 0,C 180,E1 -1358.255,E2 -1358.255} C_VEL
LIN {X 0,Y 587.345,Z 132.82,A -85,B 0,C 180,E1 -1361.134,E2 -1361.134} C_VEL
LIN {X 0,Y 587.362,Z 132.817,A -85,B 0,C 180,E1 -1364.26,E2 -1364.26} C_VEL
LIN {X 0,Y 587.347,Z 132.825,A -85,B 0,C 180,E1 -1367.406,E2 -1367.406} C_VEL
LIN {X 0,Y 587.328,Z 132.82,A -85,B 0,C 180,E1 -1370.305,E2 -1370.305} C_VEL
LIN {X 0,Y 587.319,Z 132.829,A -85,B 0,C 180,E1 -1373.259,E2 -1373.259} C_VEL
LIN {X 0,Y 587.331,Z 132.826,A -85,B 0,C 180,E1 -1375.517,E2 -1375.517} C_VEL
LIN {X 0,Y 587.345,Z 132.819,A -85,B 0,C 180,E1 -1377.818,E2 -1377.818} C_VEL
LIN {X 0,Y 587.348,Z 132.817,A -85,B 0,C 180,E1 -1380.512,E2 -1380.512} C_VEL
LIN {X 0,Y 587.331,Z 132.823,A -85,B 0,C 180,E1 -1383.396,E2 -1383.396} C_VEL
LIN {X 0,Y 587.315,Z 132.82,A -85,B 0,C 180,E1 -1385.898,E2 -1385.898} C_VEL
LIN {X 0,Y 587.331,Z 132.822,A -85,B 0,C 180,E1 -1388.479,E2 -1388.479} C_VEL
LIN {X 0,Y 587.333,Z 132.821,A -85,B 0,C 180,E1 -1391.157,E2 -1391.157} C_VEL
LIN {X 0,Y 587.321,Z 132.819,A -85,B 0,C 180,E1 -1394.113,E2 -1394.113} C_VEL
LIN {X 0,Y 587.332,Z 132.825,A -85,B 0,C 180,E1 -1396.996,E2 -1396.996} C_VEL
LIN {X 0,Y 587.316,Z 132.821,A -85,B 0,C 180,E1 -1399.981,E2 -1399.981} C_VEL
LIN {X 0,Y 587.34,Z 132.824,A -85,B 0,C 180,E1 -1402.393,E2 -1402.393} C_VEL
LIN {X 0,Y 587.345,Z 132.819,A -85,B 0,C 180,E1 -1404.946,E2 -1404.946} C_VEL
LIN {X 0,Y 587.336,Z 132.818,A -85,B 0,C 180,E1 -1407.421,E2 -1407.421} C_VEL
LIN {X 0,Y 587.329,Z 132.821,A -85,B 0,C 180,E1 -1409.83,E2 -1409.83} C_VEL
LIN {X 0,Y 587.346,Z 132.825,A -85,B 0,C 180,E1 -1412.307,E2 -1412.307} C_VEL
LIN {X 0,Y 587.335,Z 132.825,A -85,B 0,C 180,E1 -1414.484,E2 -1414.484} C_VEL
LIN {X 0,Y 587.336,Z 132.819,A -85,B 0,C 180,E1 -1417.486,E2 -1417.486} C_VEL
LIN {X 0,Y 587.338,Z 132.821,A -85,B 0,C 180,E1 -1420.425,E2 -1420.425} C_VEL
LIN {X 0,Y 587.343,Z 132.817,A -85,B 0,C 180,E1 -1423.311,E2 -1423.311} C_VEL
LIN {X 0,Y 587.358,Z 132.822,A -85,B 0,C 180,E1 -1426.155,E2 -1426.155} C_VEL
LIN {X 0,Y 587.335,Z 132.817,A -85,B 0,C 180,E1 -1428.963,E2 -1428.963} C_VEL
LIN {X 0,Y 587.362,Z 132.821,A -85,B 0,C 180,E1 -1431.745,E2 -1431.745} C_VEL
LIN {X 0,Y 587.358,Z 132.816,A -85,B 0,C 180,E1 -1434.507,E2 -1434.507} C_VEL
LIN {X 0,Y 587.369,Z 132.817,A -85,B 0,C 180,E1 -1437.257,E2 -1437.257} C_VEL
LIN {X 0,Y 587.38,Z 132.814,A -85,B 0,C 180,E1 -1440,E2 -1440} C_VEL
LIN {X 0,Y 587.372,Z 132.814,A -85,B 0,C 180,E1 -1442.744,E2 -1442.744} C_VEL
LIN {X 0,Y 587.354,Z 132.826,A -85,B 0,C 180,E1 -1445.493,E2 -1445.493} C_VEL
LIN {X 0,Y 587.362,Z 132.813,A -85,B 0,C 180,E1 -1448.256,E2 -1448.256} C_VEL
LIN {X 0,Y 587.344,Z 132.822,A -85,B 0,C 180,E1 -1451.134,E2 -1451.134} C_VEL
LIN {X 0,Y 587.362,Z 132.815,A -85,B 0,C 180,E1 -1454.261,E2 -1454.261} C_VEL
LIN {X 0,Y 587.353,Z 132.82,A -85,B 0,C 180,E1 -1457.406,E2 -1457.406} C_VEL
LIN {X 0,Y 587.324,Z 132.819,A -85,B 0,C 180,E1 -1460.305,E2 -1460.305} C_VEL
LIN {X 0,Y 587.32,Z 132.826,A -85,B 0,C 180,E1 -1463.259,E2 -1463.259} C_VEL
LIN {X 0,Y 587.336,Z 132.819,A -85,B 0,C 180,E1 -1465.517,E2 -1465.517} C_VEL
LIN {X 0,Y 587.344,Z 132.816,A -85,B 0,C 180,E1 -1467.818,E2 -1467.818} C_VEL
LIN {X 0,Y 587.34,Z 132.823,A -85,B 0,C 180,E1 -1470.511,E2 -1470.511} C_VEL
LIN {X 0,Y 587.334,Z 132.818,A -85,B 0,C 180,E1 -1473.397,E2 -1473.397} C_VEL
LIN {X 0,Y 587.292,Z 132.824,A -85,B 0,C 180,E1 -1475.9,E2 -1475.9} C_VEL
LIN {X 0,Y 587.326,Z 132.828,A -85,B 0,C 180,E1 -1478.48,E2 -1478.48} C_VEL
LIN {X 0,Y 587.335,Z 132.82,A -85,B 0,C 180,E1 -1481.157,E2 -1481.157} C_VEL
LIN {X 0,Y 587.326,Z 132.824,A -85,B 0,C 180,E1 -1484.114,E2 -1484.114} C_VEL
LIN {X 0,Y 587.312,Z 132.823,A -85,B 0,C 180,E1 -1486.994,E2 -1486.994} C_VEL
LIN {X 0,Y 587.317,Z 132.821,A -85,B 0,C 180,E1 -1489.746,E2 -1489.746} C_VEL
LIN {X 0,Y 587.345,Z 132.825,A -85,B 0,C 180,E1 -1492.393,E2 -1492.393} C_VEL
LIN {X 0,Y 587.347,Z 132.819,A -85,B 0,C 180,E1 -1495.653,E2 -1495.653} C_VEL
LIN {X 0,Y 587.35,Z 132.825,A -85,B 0,C 180,E1 -1498.232,E2 -1498.232} C_VEL
LIN {X 0,Y 587.347,Z 132.818,A -85,B 0,C 180,E1 -1500.868,E2 -1500.868} C_VEL
LIN {X 0,Y 587.36,Z 132.824,A -85,B 0,C 180,E1 -1503.82,E2 -1503.82} C_VEL
LIN {X 0,Y 587.35,Z 132.968,A -85,B 0,C 180,E1 -1505.421,E2 -1505.421} C_VEL
LIN {X 0,Y 587.722,Z 136.049,A -85,B 0,C 180,E1 -1506.011,E2 -1506.011} C_VEL
LIN {X 0,Y 587.573,Z 152.742,A -85,B 0,C 180,E1 -1508.972,E2 -1508.972} C_VEL
LIN {X 0,Y 587.48,Z 167.229,A -85,B 0,C 180,E1 -1511.518,E2 -1511.518} C_VEL
LIN {X 0,Y 587.4,Z 182.75,A -85,B 0,C 180,E1 -1514.205,E2 -1514.205} C_VEL
LIN {X 0,Y 587.388,Z 196.24,A -85,B 0,C 180,E1 -1516.486,E2 -1516.486} C_VEL
LIN {X 0,Y 587.711,Z 198.731,A -85,B 0,C 180,E1 -1516.559,E2 -1516.559} C_VEL
LIN {X 0,Y 587.728,Z 302.749,A -85,B 0,C 180,E1 -1517.855,E2 -1517.855} C_VEL
LIN {X 0,Y 587.68,Z 315.506,A -85,B 0,C 180,E1 -1518.139,E2 -1518.139} C_VEL
LIN {X 0,Y 587.609,Z 328.821,A -85,B 0,C 180,E1 -1518.592,E2 -1518.592} C_VEL
LIN {X 0,Y 587.555,Z 340.558,A -85,B 0,C 180,E1 -1519.141,E2 -1519.141} C_VEL
LIN {X 0,Y 587.441,Z 350.875,A -85,B 0,C 180,E1 -1519.749,E2 -1519.749} C_VEL
LIN {X 0,Y 587.381,Z 361.549,A -85,B 0,C 180,E1 -1520.531,E2 -1520.531} C_VEL
LIN {X 0,Y 587.322,Z 371.12,A -85,B 0,C 180,E1 -1521.398,E2 -1521.398} C_VEL
LIN {X 0,Y 587.273,Z 378.934,A -85,B 0,C 180,E1 -1522.263,E2 -1522.263} C_VEL
LIN {X 0,Y 587.229,Z 385.448,A -85,B 0,C 180,E1 -1523.126,E2 -1523.126} C_VEL
LIN {X 0,Y 587.23,Z 391.832,A -85,B 0,C 180,E1 -1524.161,E2 -1524.161} C_VEL
LIN {X 0,Y 587.146,Z 396.927,A -85,B 0,C 180,E1 -1525.194,E2 -1525.194} C_VEL
LIN {X 0,Y 587.213,Z 400.878,A -85,B 0,C 180,E1 -1526.226,E2 -1526.226} C_VEL
LIN {X 0,Y 587.132,Z 403.791,A -85,B 0,C 180,E1 -1527.256,E2 -1527.256} C_VEL
LIN {X 0,Y 587.147,Z 406.19,A -85,B 0,C 180,E1 -1528.628,E2 -1528.628} C_VEL
LIN {X 0,Y 587.14,Z 406.782,A -85,B 0,C 180,E1 -1529.314,E2 -1529.314} C_VEL
LIN {X 0,Y 587.14,Z 406.782,A -85,B 0,C 180,E1 -1530.686,E2 -1530.686} C_VEL
LIN {X 0,Y 587.147,Z 406.19,A -85,B 0,C 180,E1 -1531.372,E2 -1531.372} C_VEL
LIN {X 0,Y 587.132,Z 403.791,A -85,B 0,C 180,E1 -1532.744,E2 -1532.744} C_VEL
LIN {X 0,Y 587.213,Z 400.878,A -85,B 0,C 180,E1 -1533.774,E2 -1533.774} C_VEL
LIN {X 0,Y 587.146,Z 396.927,A -85,B 0,C 180,E1 -1534.806,E2 -1534.806} C_VEL
LIN {X 0,Y 587.23,Z 391.832,A -85,B 0,C 180,E1 -1535.839,E2 -1535.839} C_VEL
LIN {X 0,Y 587.229,Z 385.448,A -85,B 0,C 180,E1 -1536.874,E2 -1536.874} C_VEL
LIN {X 0,Y 587.287,Z 377.492,A -85,B 0,C 180,E1 -1537.91,E2 -1537.91} C_VEL
LIN {X 0,Y 587.335,Z 369.351,A -85,B 0,C 180,E1 -1538.776,E2 -1538.776} C_VEL
LIN {X 0,Y 587.389,Z 359.349,A -85,B 0,C 180,E1 -1539.643,E2 -1539.643} C_VEL
LIN {X 0,Y 587.464,Z 349.526,A -85,B 0,C 180,E1 -1540.338,E2 -1540.338} C_VEL
LIN {X 0,Y 587.552,Z 338.928,A -85,B 0,C 180,E1 -1540.946,E2 -1540.946} C_VEL
LIN {X 0,Y 587.616,Z 325.234,A -85,B 0,C 180,E1 -1541.547,E2 -1541.547} C_VEL
LIN {X 0,Y 587.688,Z 312.948,A -85,B 0,C 180,E1 -1541.927,E2 -1541.927} C_VEL
LIN {X 0,Y 587.733,Z 301.418,A -85,B 0,C 180,E1 -1542.167,E2 -1542.167} C_VEL
LIN {X 0,Y 587.727,Z 198.731,A -85,B 0,C 180,E1 -1543.44,E2 -1543.44} C_VEL
LIN {X 0,Y 587.388,Z 196.24,A -85,B 0,C 180,E1 -1543.514,E2 -1543.514} C_VEL
LIN {X 0,Y 587.441,Z 180.681,A -85,B 0,C 180,E1 -1546.15,E2 -1546.15} C_VEL
LIN {X 0,Y 587.52,Z 165.159,A -85,B 0,C 180,E1 -1548.843,E2 -1548.843} C_VEL
LIN {X 0,Y 587.638,Z 149.638,A -85,B 0,C 180,E1 -1551.577,E2 -1551.577} C_VEL
LIN {X 0,Y 587.668,Z 134.477,A -85,B 0,C 180,E1 -1554.278,E2 -1554.278} C_VEL
LIN {X 0,Y 587.363,Z 132.868,A -85,B 0,C 180,E1 -1554.629,E2 -1554.629} C_VEL
LIN {X 0,Y 587.329,Z 132.821,A -85,B 0,C 180,E1 -1557.046,E2 -1557.046} C_VEL
LIN {X 0,Y 587.344,Z 132.82,A -85,B 0,C 180,E1 -1559.379,E2 -1559.379} C_VEL
LIN {X 0,Y 587.353,Z 132.826,A -85,B 0,C 180,E1 -1561.836,E2 -1561.836} C_VEL
LIN {X 0,Y 587.347,Z 132.819,A -85,B 0,C 180,E1 -1564.347,E2 -1564.347} C_VEL
LIN {X 0,Y 587.345,Z 132.825,A -85,B 0,C 180,E1 -1567.607,E2 -1567.607} C_VEL
LIN {X 0,Y 587.316,Z 132.821,A -85,B 0,C 180,E1 -1570.254,E2 -1570.254} C_VEL
LIN {X 0,Y 587.314,Z 132.824,A -85,B 0,C 180,E1 -1573.118,E2 -1573.118} C_VEL
LIN {X 0,Y 587.322,Z 132.823,A -85,B 0,C 180,E1 -1576.049,E2 -1576.049} C_VEL
LIN {X 0,Y 587.335,Z 132.821,A -85,B 0,C 180,E1 -1578.924,E2 -1578.924} C_VEL
LIN {X 0,Y 587.326,Z 132.828,A -85,B 0,C 180,E1 -1581.52,E2 -1581.52} C_VEL
LIN {X 0,Y 587.292,Z 132.824,A -85,B 0,C 180,E1 -1584.1,E2 -1584.1} C_VEL
LIN {X 0,Y 587.334,Z 132.818,A -85,B 0,C 180,E1 -1586.603,E2 -1586.603} C_VEL
LIN {X 0,Y 587.34,Z 132.823,A -85,B 0,C 180,E1 -1589.489,E2 -1589.489} C_VEL
LIN {X 0,Y 587.349,Z 132.816,A -85,B 0,C 180,E1 -1592.307,E2 -1592.307} C_VEL
LIN {X 0,Y 587.336,Z 132.819,A -85,B 0,C 180,E1 -1594.483,E2 -1594.483} C_VEL
LIN {X 0,Y 587.336,Z 132.82,A -85,B 0,C 180,E1 -1597.486,E2 -1597.486} C_VEL
LIN {X 0,Y 587.34,Z 132.819,A -85,B 0,C 180,E1 -1600.425,E2 -1600.425} C_VEL
LIN {X 0,Y 587.341,Z 132.82,A -85,B 0,C 180,E1 -1603.311,E2 -1603.311} C_VEL
LIN {X 0,Y 587.359,Z 132.817,A -85,B 0,C 180,E1 -1606.154,E2 -1606.154} C_VEL
LIN {X 0,Y 587.335,Z 132.821,A -85,B 0,C 180,E1 -1608.962,E2 -1608.962} C_VEL
LIN {X 0,Y 587.362,Z 132.813,A -85,B 0,C 180,E1 -1611.744,E2 -1611.744} C_VEL
LIN {X 0,Y 587.354,Z 132.826,A -85,B 0,C 180,E1 -1614.507,E2 -1614.507} C_VEL
LIN {X 0,Y 587.372,Z 132.814,A -85,B 0,C 180,E1 -1617.256,E2 -1617.256} C_VEL
LIN {X 0,Y 587.38,Z 132.814,A -85,B 0,C 180,E1 -1620,E2 -1620} C_VEL
LIN {X 0,Y 587.369,Z 132.817,A -85,B 0,C 180,E1 -1622.743,E2 -1622.743} C_VEL
LIN {X 0,Y 587.358,Z 132.816,A -85,B 0,C 180,E1 -1625.493,E2 -1625.493} C_VEL
LIN {X 0,Y 587.362,Z 132.821,A -85,B 0,C 180,E1 -1628.255,E2 -1628.255} C_VEL
LIN {X 0,Y 587.343,Z 132.816,A -85,B 0,C 180,E1 -1631.133,E2 -1631.133} C_VEL
LIN {X 0,Y 587.361,Z 132.821,A -85,B 0,C 180,E1 -1634.261,E2 -1634.261} C_VEL
LIN {X 0,Y 587.355,Z 132.818,A -85,B 0,C 180,E1 -1637.405,E2 -1637.405} C_VEL
LIN {X 0,Y 587.321,Z 132.821,A -85,B 0,C 180,E1 -1638.306,E2 -1638.306} C_VEL
LIN {X 0,Y 586.665,Z 132.901,A -85,B 0,C 180,E1 -1638.878,E2 -1638.878} C_VEL
LIN {X 0,Y 583.833,Z 133.261,A -85,B 0,C 180,E1 -1639.806,E2 -1639.806} C_VEL
LIN {X 0,Y 581.424,Z 133.56,A -85,B 0,C 180,E1 -1640.553,E2 -1640.553} C_VEL
LIN {X 0,Y 580.373,Z 133.687,A -85,B 0,C 180,E1 -1641.129,E2 -1641.129} C_VEL
LIN {X 0,Y 580.278,Z 133.699,A -85,B 0,C 180,E1 -1641.325,E2 -1641.325} C_VEL
LIN {X 0,Y 580.275,Z 133.705,A -85,B 0,C 180,E1 -1643.558,E2 -1643.558} C_VEL
LIN {X 0,Y 580.324,Z 133.691,A -85,B 0,C 180,E1 -1646.341,E2 -1646.341} C_VEL
LIN {X 0,Y 580.298,Z 133.699,A -85,B 0,C 180,E1 -1649.31,E2 -1649.31} C_VEL
LIN {X 0,Y 580.298,Z 133.696,A -85,B 0,C 180,E1 -1652.2,E2 -1652.2} C_VEL
LIN {X 0,Y 580.296,Z 133.693,A -85,B 0,C 180,E1 -1654.695,E2 -1654.695} C_VEL
LIN {X 0,Y 580.295,Z 133.703,A -85,B 0,C 180,E1 -1657.268,E2 -1657.268} C_VEL
LIN {X 0,Y 580.292,Z 133.694,A -85,B 0,C 180,E1 -1660.271,E2 -1660.271} C_VEL
LIN {X 0,Y 580.286,Z 133.698,A -85,B 0,C 180,E1 -1662.705,E2 -1662.705} C_VEL
LIN {X 0,Y 580.265,Z 133.7,A -85,B 0,C 180,E1 -1665.609,E2 -1665.609} C_VEL
LIN {X 0,Y 580.294,Z 133.691,A -85,B 0,C 180,E1 -1668.233,E2 -1668.233} C_VEL
LIN {X 0,Y 580.287,Z 133.704,A -85,B 0,C 180,E1 -1670.966,E2 -1670.966} C_VEL
LIN {X 0,Y 580.292,Z 133.696,A -85,B 0,C 180,E1 -1673.599,E2 -1673.599} C_VEL
LIN {X 0,Y 580.315,Z 133.691,A -85,B 0,C 180,E1 -1676.146,E2 -1676.146} C_VEL
LIN {X 0,Y 580.286,Z 133.703,A -85,B 0,C 180,E1 -1678.616,E2 -1678.616} C_VEL
LIN {X 0,Y 580.29,Z 133.702,A -85,B 0,C 180,E1 -1681.024,E2 -1681.024} C_VEL
LIN {X 0,Y 580.288,Z 133.697,A -85,B 0,C 180,E1 -1683.666,E2 -1683.666} C_VEL
LIN {X 0,Y 580.297,Z 133.696,A -85,B 0,C 180,E1 -1685.684,E2 -1685.684} C_VEL
LIN {X 0,Y 580.272,Z 133.7,A -85,B 0,C 180,E1 -1687.948,E2 -1687.948} C_VEL
LIN {X 0,Y 580.315,Z 133.697,A -85,B 0,C 180,E1 -1690.914,E2 -1690.914} C_VEL
LIN {X 0,Y 580.277,Z 133.7,A -85,B 0,C 180,E1 -1693.826,E2 -1693.826} C_VEL
LIN {X 0,Y 580.322,Z 133.697,A -85,B 0,C 180,E1 -1695.983,E2 -1695.983} C_VEL
LIN {X 0,Y 580.301,Z 133.698,A -85,B 0,C 180,E1 -1698.827,E2 -1698.827} C_VEL
LIN {X 0,Y 580.332,Z 133.694,A -85,B 0,C 180,E1 -1701.644,E2 -1701.644} C_VEL
LIN {X 0,Y 580.323,Z 133.698,A -85,B 0,C 180,E1 -1704.44,E2 -1704.44} C_VEL
LIN {X 0,Y 580.336,Z 133.691,A -85,B 0,C 180,E1 -1707.223,E2 -1707.223} C_VEL
LIN {X 0,Y 580.352,Z 133.699,A -85,B 0,C 180,E1 -1710,E2 -1710} C_VEL
LIN {X 0,Y 580.336,Z 133.691,A -85,B 0,C 180,E1 -1712.777,E2 -1712.777} C_VEL
LIN {X 0,Y 580.323,Z 133.698,A -85,B 0,C 180,E1 -1715.56,E2 -1715.56} C_VEL
LIN {X 0,Y 580.332,Z 133.694,A -85,B 0,C 180,E1 -1718.356,E2 -1718.356} C_VEL
LIN {X 0,Y 580.297,Z 133.698,A -85,B 0,C 180,E1 -1721.191,E2 -1721.191} C_VEL
LIN {X 0,Y 580.322,Z 133.697,A -85,B 0,C 180,E1 -1724.017,E2 -1724.017} C_VEL
LIN {X 0,Y 580.309,Z 133.696,A -85,B 0,C 180,E1 -1726.914,E2 -1726.914} C_VEL
LIN {X 0,Y 580.303,Z 133.7,A -85,B 0,C 180,E1 -1729.822,E2 -1729.822} C_VEL
LIN {X 0,Y 580.292,Z 133.698,A -85,B 0,C 180,E1 -1732.802,E2 -1732.802} C_VEL
LIN {X 0,Y 580.303,Z 133.701,A -85,B 0,C 180,E1 -1735.08,E2 -1735.08} C_VEL
LIN {X 0,Y 580.297,Z 133.695,A -85,B 0,C 180,E1 -1738.185,E2 -1738.185} C_VEL
LIN {X 0,Y 580.296,Z 133.697,A -85,B 0,C 180,E1 -1740.697,E2 -1740.697} C_VEL
LIN {X 0,Y 580.3,Z 133.699,A -85,B 0,C 180,E1 -1743.317,E2 -1743.317} C_VEL
LIN {X 0,Y 580.272,Z 133.698,A -85,B 0,C 180,E1 -1745.761,E2 -1745.761} C_VEL
LIN {X 0,Y 580.286,Z 133.697,A -85,B 0,C 180,E1 -1748.146,E2 -1748.146} C_VEL
LIN {X 0,Y 580.296,Z 133.702,A -85,B 0,C 180,E1 -1750.843,E2 -1750.843} C_VEL
LIN {X 0,Y 580.274,Z 133.696,A -85,B 0,C 180,E1 -1753.658,E2 -1753.658} C_VEL
LIN {X 0,Y 580.288,Z 133.704,A -85,B 0,C 180,E1 -1756.608,E2 -1756.608} C_VEL
LIN {X 0,Y 580.296,Z 133.697,A -85,B 0,C 180,E1 -1759.157,E2 -1759.157} C_VEL
LIN {X 0,Y 580.285,Z 133.698,A -85,B 0,C 180,E1 -1761.927,E2 -1761.927} C_VEL
LIN {X 0,Y 580.301,Z 133.703,A -85,B 0,C 180,E1 -1764.457,E2 -1764.457} C_VEL
LIN {X 0,Y 580.287,Z 133.699,A -85,B 0,C 180,E1 -1766.975,E2 -1766.975} C_VEL
LIN {X 0,Y 580.297,Z 133.695,A -85,B 0,C 180,E1 -1769.426,E2 -1769.426} C_VEL
LIN {X 0,Y 580.315,Z 133.698,A -85,B 0,C 180,E1 -1772.137,E2 -1772.137} C_VEL
LIN {X 0,Y 580.304,Z 133.695,A -85,B 0,C 180,E1 -1774.921,E2 -1774.921} C_VEL
LIN {X 0,Y 580.269,Z 133.704,A -85,B 0,C 180,E1 -1777.948,E2 -1777.948} C_VEL
LIN {X 0,Y 580.314,Z 133.69,A -85,B 0,C 180,E1 -1780.914,E2 -1780.914} C_VEL
LIN {X 0,Y 580.276,Z 133.703,A -85,B 0,C 180,E1 -1783.826,E2 -1783.826} C_VEL
LIN {X 0,Y 580.323,Z 133.702,A -85,B 0,C 180,E1 -1785.983,E2 -1785.983} C_VEL
LIN {X 0,Y 580.3,Z 133.693,A -85,B 0,C 180,E1 -1788.827,E2 -1788.827} C_VEL
LIN {X 0,Y 580.325,Z 133.695,A -85,B 0,C 180,E1 -1791.644,E2 -1791.644} C_VEL
LIN {X 0,Y 580.323,Z 133.693,A -85,B 0,C 180,E1 -1794.441,E2 -1794.441} C_VEL
LIN {X 0,Y 580.335,Z 133.693,A -85,B 0,C 180,E1 -1797.224,E2 -1797.224} C_VEL
LIN {X 0,Y 580.349,Z 133.69,A -85,B 0,C 180,E1 -1800,E2 -1800} C_VEL
LIN {X 0,Y 580.338,Z 133.69,A -85,B 0,C 180,E1 -1802.777,E2 -1802.777} C_VEL
LIN {X 0,Y 580.32,Z 133.7,A -85,B 0,C 180,E1 -1805.56,E2 -1805.56} C_VEL
LIN {X 0,Y 580.325,Z 133.689,A -85,B 0,C 180,E1 -1808.356,E2 -1808.356} C_VEL
LIN {X 0,Y 580.296,Z 133.7,A -85,B 0,C 180,E1 -1811.191,E2 -1811.191} C_VEL
LIN {X 0,Y 580.324,Z 133.692,A -85,B 0,C 180,E1 -1814.017,E2 -1814.017} C_VEL
LIN {X 0,Y 580.309,Z 133.698,A -85,B 0,C 180,E1 -1816.914,E2 -1816.914} C_VEL
LIN {X 0,Y 580.301,Z 133.694,A -85,B 0,C 180,E1 -1819.823,E2 -1819.823} C_VEL
LIN {X 0,Y 580.292,Z 133.702,A -85,B 0,C 180,E1 -1822.803,E2 -1822.803} C_VEL
LIN {X 0,Y 580.306,Z 133.7,A -85,B 0,C 180,E1 -1825.08,E2 -1825.08} C_VEL
LIN {X 0,Y 580.296,Z 133.695,A -85,B 0,C 180,E1 -1828.186,E2 -1828.186} C_VEL
LIN {X 0,Y 580.291,Z 133.704,A -85,B 0,C 180,E1 -1830.697,E2 -1830.697} C_VEL
LIN {X 0,Y 580.303,Z 133.694,A -85,B 0,C 180,E1 -1833.317,E2 -1833.317} C_VEL
LIN {X 0,Y 580.248,Z 133.701,A -85,B 0,C 180,E1 -1835.757,E2 -1835.757} C_VEL
LIN {X 0,Y 580.285,Z 133.7,A -85,B 0,C 180,E1 -1838.147,E2 -1838.147} C_VEL
LIN {X 0,Y 580.297,Z 133.7,A -85,B 0,C 180,E1 -1840.844,E2 -1840.844} C_VEL
LIN {X 0,Y 580.278,Z 133.698,A -85,B 0,C 180,E1 -1843.658,E2 -1843.658} C_VEL
LIN {X 0,Y 580.273,Z 133.705,A -85,B 0,C 180,E1 -1846.61,E2 -1846.61} C_VEL
LIN {X 0,Y 580.299,Z 133.693,A -85,B 0,C 180,E1 -1849.157,E2 -1849.157} C_VEL
LIN {X 0,Y 580.29,Z 133.701,A -85,B 0,C 180,E1 -1851.928,E2 -1851.928} C_VEL
LIN {X 0,Y 580.253,Z 133.706,A -85,B 0,C 180,E1 -1854.453,E2 -1854.453} C_VEL
LIN {X 0,Y 580.29,Z 133.696,A -85,B 0,C 180,E1 -1856.976,E2 -1856.976} C_VEL
LIN {X 0,Y 580.303,Z 133.697,A -85,B 0,C 180,E1 -1859.426,E2 -1859.426} C_VEL
LIN {X 0,Y 580.3,Z 133.703,A -85,B 0,C 180,E1 -1862.142,E2 -1862.142} C_VEL
LIN {X 0,Y 580.337,Z 133.767,A -85,B 0,C 180,E1 -1865.255,E2 -1865.255} C_VEL
LIN {X 0,Y 580.756,Z 138.037,A -85,B 0,C 180,E1 -1866.084,E2 -1866.084} C_VEL
LIN {X 0,Y 580.609,Z 154.888,A -85,B 0,C 180,E1 -1869.105,E2 -1869.105} C_VEL
LIN {X 0,Y 580.488,Z 170.333,A -85,B 0,C 180,E1 -1871.835,E2 -1871.835} C_VEL
LIN {X 0,Y 580.349,Z 186.89,A -85,B 0,C 180,E1 -1874.729,E2 -1874.729} C_VEL
LIN {X 0,Y 580.361,Z 196.249,A -85,B 0,C 180,E1 -1876.319,E2 -1876.319} C_VEL
LIN {X 0,Y 580.678,Z 198.731,A -85,B 0,C 180,E1 -1876.394,E2 -1876.394} C_VEL
LIN {X 0,Y 580.946,Z 207.675,A -85,B 0,C 180,E1 -1876.511,E2 -1876.511} C_VEL
LIN {X 0,Y 580.81,Z 302.683,A -85,B 0,C 180,E1 -1877.708,E2 -1877.708} C_VEL
LIN {X 0,Y 580.767,Z 314.656,A -85,B 0,C 180,E1 -1877.973,E2 -1877.973} C_VEL
LIN {X 0,Y 580.677,Z 328.401,A -85,B 0,C 180,E1 -1878.437,E2 -1878.437} C_VEL
LIN {X 0,Y 580.572,Z 338.907,A -85,B 0,C 180,E1 -1878.921,E2 -1878.921} C_VEL
LIN {X 0,Y 580.462,Z 349.507,A -85,B 0,C 180,E1 -1879.536,E2 -1879.536} C_VEL
LIN {X 0,Y 580.369,Z 359.333,A -85,B 0,C 180,E1 -1880.239,E2 -1880.239} C_VEL
LIN {X 0,Y 580.304,Z 369.355,A -85,B 0,C 180,E1 -1881.117,E2 -1881.117} C_VEL
LIN {X 0,Y 580.221,Z 378.924,A -85,B 0,C 180,E1 -1882.168,E2 -1882.168} C_VEL
LIN {X 0,Y 580.157,Z 385.436,A -85,B 0,C 180,E1 -1883.042,E2 -1883.042} C_VEL
LIN {X 0,Y 580.162,Z 391.821,A -85,B 0,C 180,E1 -1884.09,E2 -1884.09} C_VEL
LIN {X 0,Y 580.052,Z 396.917,A -85,B 0,C 180,E1 -1885.135,E2 -1885.135} C_VEL
LIN {X 0,Y 580.11,Z 400.869,A -85,B 0,C 180,E1 -1886.179,E2 -1886.179} C_VEL
LIN {X 0,Y 580.043,Z 403.785,A -85,B 0,C 180,E1 -1887.222,E2 -1887.222} C_VEL
LIN {X 0,Y 580.047,Z 406.192,A -85,B 0,C 180,E1 -1888.611,E2 -1888.611} C_VEL
LIN {X 0,Y 580.04,Z 406.781,A -85,B 0,C 180,E1 -1889.306,E2 -1889.306} C_VEL
LIN {X 0,Y 580.04,Z 406.781,A -85,B 0,C 180,E1 -1890.694,E2 -1890.694} C_VEL
LIN {X 0,Y 580.047,Z 406.192,A -85,B 0,C 180,E1 -1891.389,E2 -1891.389} C_VEL
LIN {X 0,Y 580.043,Z 403.785,A -85,B 0,C 180,E1 -1892.778,E2 -1892.778} C_VEL
LIN {X 0,Y 580.11,Z 400.869,A -85,B 0,C 180,E1 -1893.821,E2 -1893.821} C_VEL
LIN {X 0,Y 580.052,Z 396.917,A -85,B 0,C 180,E1 -1894.865,E2 -1894.865} C_VEL
LIN {X 0,Y 580.162,Z 391.821,A -85,B 0,C 180,E1 -1895.91,E2 -1895.91} C_VEL
LIN {X 0,Y 580.157,Z 385.436,A -85,B 0,C 180,E1 -1896.958,E2 -1896.958} C_VEL
LIN {X 0,Y 580.242,Z 377.496,A -85,B 0,C 180,E1 -1898.007,E2 -1898.007} C_VEL
LIN {X 0,Y 580.304,Z 369.355,A -85,B 0,C 180,E1 -1898.883,E2 -1898.883} C_VEL
LIN {X 0,Y 580.363,Z 359.333,A -85,B 0,C 180,E1 -1899.761,E2 -1899.761} C_VEL
LIN {X 0,Y 580.462,Z 349.507,A -85,B 0,C 180,E1 -1900.464,E2 -1900.464} C_VEL
LIN {X 0,Y 580.578,Z 338.907,A -85,B 0,C 180,E1 -1901.079,E2 -1901.079} C_VEL
LIN {X 0,Y 580.658,Z 326.167,A -85,B 0,C 180,E1 -1901.652,E2 -1901.652} C_VEL
LIN {X 0,Y 580.742,Z 313.782,A -85,B 0,C 180,E1 -1902.049,E2 -1902.049} C_VEL
LIN {X 0,Y 580.81,Z 302.683,A -85,B 0,C 180,E1 -1902.292,E2 -1902.292} C_VEL
LIN {X 0,Y 580.818,Z 199.402,A -85,B 0,C 180,E1 -1903.595,E2 -1903.595} C_VEL
LIN {X 0,Y 580.386,Z 196.567,A -85,B 0,C 180,E1 -1903.658,E2 -1903.658} C_VEL
LIN {X 0,Y 580.325,Z 194.133,A -85,B 0,C 180,E1 -1904.017,E2 -1904.017} C_VEL
LIN {X 0,Y 580.4,Z 178.611,A -85,B 0,C 180,E1 -1906.713,E2 -1906.713} C_VEL
LIN {X 0,Y 580.547,Z 164.355,A -85,B 0,C 180,E1 -1909.221,E2 -1909.221} C_VEL
LIN {X 0,Y 580.634,Z 149.509,A -85,B 0,C 180,E1 -1911.851,E2 -1911.851} C_VEL
LIN {X 0,Y 580.718,Z 135.974,A -85,B 0,C 180,E1 -1914.297,E2 -1914.297} C_VEL
LIN {X 0,Y 580.334,Z 133.745,A -85,B 0,C 180,E1 -1914.759,E2 -1914.759} C_VEL
LIN {X 0,Y 580.299,Z 133.703,A -85,B 0,C 180,E1 -1917.858,E2 -1917.858} C_VEL
LIN {X 0,Y 580.293,Z 133.697,A -85,B 0,C 180,E1 -1920.695,E2 -1920.695} C_VEL
LIN {X 0,Y 580.304,Z 133.696,A -85,B 0,C 180,E1 -1923.316,E2 -1923.316} C_VEL
LIN {X 0,Y 580.247,Z 133.709,A -85,B 0,C 180,E1 -1925.756,E2 -1925.756} C_VEL
LIN {X 0,Y 580.289,Z 133.7,A -85,B 0,C 180,E1 -1928.146,E2 -1928.146} C_VEL
LIN {X 0,Y 580.298,Z 133.693,A -85,B 0,C 180,E1 -1930.843,E2 -1930.843} C_VEL
LIN {X 0,Y 580.272,Z 133.707,A -85,B 0,C 180,E1 -1933.658,E2 -1933.658} C_VEL
LIN {X 0,Y 580.277,Z 133.698,A -85,B 0,C 180,E1 -1936.609,E2 -1936.609} C_VEL
LIN {X 0,Y 580.297,Z 133.7,A -85,B 0,C 180,E1 -1939.156,E2 -1939.156} C_VEL
LIN {X 0,Y 580.287,Z 133.699,A -85,B 0,C 180,E1 -1941.927,E2 -1941.927} C_VEL
LIN {X 0,Y 580.256,Z 133.7,A -85,B 0,C 180,E1 -1944.453,E2 -1944.453} C_VEL
LIN {X 0,Y 580.289,Z 133.7,A -85,B 0,C 180,E1 -1946.975,E2 -1946.975} C_VEL
LIN {X 0,Y 580.3,Z 133.701,A -85,B 0,C 180,E1 -1949.425,E2 -1949.425} C_VEL
LIN {X 0,Y 580.295,Z 133.694,A -85,B 0,C 180,E1 -1952.141,E2 -1952.141} C_VEL
LIN {X 0,Y 580.32,Z 133.698,A -85,B 0,C 180,E1 -1955.269,E2 -1955.269} C_VEL
LIN {X 0,Y 580.268,Z 133.698,A -85,B 0,C 180,E1 -1957.947,E2 -1957.947} C_VEL
LIN {X 0,Y 580.297,Z 133.701,A -85,B 0,C 180,E1 -1960.913,E2 -1960.913} C_VEL
LIN {X 0,Y 580.303,Z 133.699,A -85,B 0,C 180,E1 -1963.102,E2 -1963.102} C_VEL
LIN {X 0,Y 580.325,Z 133.692,A -85,B 0,C 180,E1 -1965.983,E2 -1965.983} C_VEL
LIN {X 0,Y 580.301,Z 133.699,A -85,B 0,C 180,E1 -1968.826,E2 -1968.826} C_VEL
LIN {X 0,Y 580.325,Z 133.689,A -85,B 0,C 180,E1 -1971.644,E2 -1971.644} C_VEL
LIN {X 0,Y 580.32,Z 133.7,A -85,B 0,C 180,E1 -1974.44,E2 -1974.44} C_VEL
LIN {X 0,Y 580.338,Z 133.69,A -85,B 0,C 180,E1 -1977.223,E2 -1977.223} C_VEL
LIN {X 0,Y 580.349,Z 133.69,A -85,B 0,C 180,E1 -1980,E2 -1980} C_VEL
LIN {X 0,Y 580.335,Z 133.693,A -85,B 0,C 180,E1 -1982.776,E2 -1982.776} C_VEL
LIN {X 0,Y 580.323,Z 133.693,A -85,B 0,C 180,E1 -1985.559,E2 -1985.559} C_VEL
LIN {X 0,Y 580.325,Z 133.695,A -85,B 0,C 180,E1 -1988.356,E2 -1988.356} C_VEL
LIN {X 0,Y 580.295,Z 133.693,A -85,B 0,C 180,E1 -1991.191,E2 -1991.191} C_VEL
LIN {X 0,Y 580.323,Z 133.702,A -85,B 0,C 180,E1 -1994.017,E2 -1994.017} C_VEL
LIN {X 0,Y 580.307,Z 133.693,A -85,B 0,C 180,E1 -1996.914,E2 -1996.914} C_VEL
LIN {X 0,Y 580.3,Z 133.701,A -85,B 0,C 180,E1 -1999.822,E2 -1999.822} C_VEL
LIN {X 0,Y 580.278,Z 133.699,A -85,B 0,C 180,E1 -2001.325,E2 -2001.325} C_VEL
LIN {X 0,Y 579.582,Z 133.793,A -85,B 0,C 180,E1 -2001.904,E2 -2001.904} C_VEL
LIN {X 0,Y 576.706,Z 134.147,A -85,B 0,C 180,E1 -2002.844,E2 -2002.844} C_VEL
LIN {X 0,Y 574.311,Z 134.448,A -85,B 0,C 180,E1 -2003.6,E2 -2003.6} C_VEL
LIN {X 0,Y 573.312,Z 134.568,A -85,B 0,C 180,E1 -2004.184,E2 -2004.184} C_VEL
LIN {X 0,Y 573.245,Z 134.575,A -85,B 0,C 180,E1 -2004.381,E2 -2004.381} C_VEL
LIN {X 0,Y 573.26,Z 134.57,A -85,B 0,C 180,E1 -2006.975,E2 -2006.975} C_VEL
LIN {X 0,Y 573.243,Z 134.581,A -85,B 0,C 180,E1 -2009.488,E2 -2009.488} C_VEL
LIN {X 0,Y 573.251,Z 134.574,A -85,B 0,C 180,E1 -2012.229,E2 -2012.229} C_VEL
LIN {X 0,Y 573.247,Z 134.572,A -85,B 0,C 180,E1 -2014.774,E2 -2014.774} C_VEL
LIN {X 0,Y 573.249,Z 134.579,A -85,B 0,C 180,E1 -2017.166,E2 -2017.166} C_VEL
LIN {X 0,Y 573.242,Z 134.578,A -85,B 0,C 180,E1 -2019.607,E2 -2019.607} C_VEL
LIN {X 0,Y 573.246,Z 134.575,A -85,B 0,C 180,E1 -2022.643,E2 -2022.643} C_VEL
LIN {X 0,Y 573.23,Z 134.576,A -85,B 0,C 180,E1 -2025.667,E2 -2025.667} C_VEL
LIN {X 0,Y 573.235,Z 134.571,A -85,B 0,C 180,E1 -2028.544,E2 -2028.544} C_VEL
LIN {X 0,Y 573.246,Z 134.579,A -85,B 0,C 180,E1 -2031.299,E2 -2031.299} C_VEL
LIN {X 0,Y 573.26,Z 134.571,A -85,B 0,C 180,E1 -2034.011,E2 -2034.011} C_VEL
LIN {X 0,Y 573.281,Z 134.571,A -85,B 0,C 180,E1 -2036.519,E2 -2036.519} C_VEL
LIN {X 0,Y 573.24,Z 134.578,A -85,B 0,C 180,E1 -2039.115,E2 -2039.115} C_VEL
LIN {X 0,Y 573.249,Z 134.573,A -85,B 0,C 180,E1 -2041.971,E2 -2041.971} C_VEL
LIN {X 0,Y 573.251,Z 134.582,A -85,B 0,C 180,E1 -2044.59,E2 -2044.59} C_VEL
LIN {X 0,Y 573.235,Z 134.576,A -85,B 0,C 180,E1 -2047.662,E2 -2047.662} C_VEL
LIN {X 0,Y 573.275,Z 134.577,A -85,B 0,C 180,E1 -2050.728,E2 -2050.728} C_VEL
LIN {X 0,Y 573.249,Z 134.574,A -85,B 0,C 180,E1 -2053.622,E2 -2053.622} C_VEL
LIN {X 0,Y 573.27,Z 134.573,A -85,B 0,C 180,E1 -2055.807,E2 -2055.807} C_VEL
LIN {X 0,Y 573.259,Z 134.576,A -85,B 0,C 180,E1 -2058.745,E2 -2058.745} C_VEL
LIN {X 0,Y 573.287,Z 134.57,A -85,B 0,C 180,E1 -2061.541,E2 -2061.541} C_VEL
LIN {X 0,Y 573.29,Z 134.575,A -85,B 0,C 180,E1 -2064.372,E2 -2064.372} C_VEL
LIN {X 0,Y 573.313,Z 134.573,A -85,B 0,C 180,E1 -2067.892,E2 -2067.892} C_VEL
LIN {X 0,Y 573.33,Z 134.565,A -85,B 0,C 180,E1 -2070.702,E2 -2070.702} C_VEL
LIN {X 0,Y 573.303,Z 134.568,A -85,B 0,C 180,E1 -2072.811,E2 -2072.811} C_VEL
LIN {X 0,Y 573.29,Z 134.575,A -85,B 0,C 180,E1 -2075.628,E2 -2075.628} C_VEL
LIN {X 0,Y 573.287,Z 134.57,A -85,B 0,C 180,E1 -2078.459,E2 -2078.459} C_VEL
LIN {X 0,Y 573.269,Z 134.576,A -85,B 0,C 180,E1 -2081.312,E2 -2081.312} C_VEL
LIN {X 0,Y 573.27,Z 134.573,A -85,B 0,C 180,E1 -2084.193,E2 -2084.193} C_VEL
LIN {X 0,Y 573.255,Z 134.577,A -85,B 0,C 180,E1 -2087.112,E2 -2087.112} C_VEL
LIN {X 0,Y 573.25,Z 134.575,A -85,B 0,C 180,E1 -2090.076,E2 -2090.076} C_VEL
LIN {X 0,Y 573.23,Z 134.581,A -85,B 0,C 180,E1 -2093.099,E2 -2093.099} C_VEL
LIN {X 0,Y 573.251,Z 134.582,A -85,B 0,C 180,E1 -2095.41,E2 -2095.41} C_VEL
LIN {X 0,Y 573.26,Z 134.572,A -85,B 0,C 180,E1 -2098.031,E2 -2098.031} C_VEL
LIN {X 0,Y 573.24,Z 134.578,A -85,B 0,C 180,E1 -2100.885,E2 -2100.885} C_VEL
LIN {X 0,Y 573.257,Z 134.573,A -85,B 0,C 180,E1 -2103.524,E2 -2103.524} C_VEL
LIN {X 0,Y 573.24,Z 134.573,A -85,B 0,C 180,E1 -2106.049,E2 -2106.049} C_VEL
LIN {X 0,Y 573.246,Z 134.579,A -85,B 0,C 180,E1 -2108.701,E2 -2108.701} C_VEL
LIN {X 0,Y 573.239,Z 134.569,A -85,B 0,C 180,E1 -2111.595,E2 -2111.595} C_VEL
LIN {X 0,Y 573.23,Z 134.576,A -85,B 0,C 180,E1 -2114.333,E2 -2114.333} C_VEL
LIN {X 0,Y 573.246,Z 134.575,A -85,B 0,C 180,E1 -2117.357,E2 -2117.357} C_VEL
LIN {X 0,Y 573.242,Z 134.578,A -85,B 0,C 180,E1 -2120.393,E2 -2120.393} C_VEL
LIN {X 0,Y 573.251,Z 134.575,A -85,B 0,C 180,E1 -2123.078,E2 -2123.078} C_VEL
LIN {X 0,Y 573.269,Z 134.568,A -85,B 0,C 180,E1 -2125.672,E2 -2125.672} C_VEL
LIN {X 0,Y 573.244,Z 134.579,A -85,B 0,C 180,E1 -2128.185,E2 -2128.185} C_VEL
LIN {X 0,Y 573.261,Z 134.576,A -85,B 0,C 180,E1 -2130.634,E2 -2130.634} C_VEL
LIN {X 0,Y 573.265,Z 134.569,A -85,B 0,C 180,E1 -2133.501,E2 -2133.501} C_VEL
LIN {X 0,Y 573.227,Z 134.584,A -85,B 0,C 180,E1 -2136.135,E2 -2136.135} C_VEL
LIN {X 0,Y 573.245,Z 134.572,A -85,B 0,C 180,E1 -2139.174,E2 -2139.174} C_VEL
LIN {X 0,Y 573.233,Z 134.572,A -85,B 0,C 180,E1 -2141.412,E2 -2141.412} C_VEL
LIN {X 0,Y 573.247,Z 134.576,A -85,B 0,C 180,E1 -2143.622,E2 -2143.622} C_VEL
LIN {X 0,Y 573.27,Z 134.577,A -85,B 0,C 180,E1 -2145.807,E2 -2145.807} C_VEL
LIN {X 0,Y 573.258,Z 134.57,A -85,B 0,C 180,E1 -2148.745,E2 -2148.745} C_VEL
LIN {X 0,Y 573.281,Z 134.571,A -85,B 0,C 180,E1 -2151.541,E2 -2151.541} C_VEL
LIN {X 0,Y 573.289,Z 134.57,A -85,B 0,C 180,E1 -2154.372,E2 -2154.372} C_VEL
LIN {X 0,Y 573.305,Z 134.57,A -85,B 0,C 180,E1 -2157.893,E2 -2157.893} C_VEL
LIN {X 0,Y 573.329,Z 134.56,A -85,B 0,C 180,E1 -2160.703,E2 -2160.703} C_VEL
LIN {X 0,Y 573.233,Z 134.584,A -85,B 0,C 180,E1 -2163.515,E2 -2163.515} C_VEL
LIN {X 0,Y 573.287,Z 134.575,A -85,B 0,C 180,E1 -2165.629,E2 -2165.629} C_VEL
LIN {X 0,Y 573.281,Z 134.566,A -85,B 0,C 180,E1 -2168.46,E2 -2168.46} C_VEL
LIN {X 0,Y 573.268,Z 134.577,A -85,B 0,C 180,E1 -2171.312,E2 -2171.312} C_VEL
LIN {X 0,Y 573.271,Z 134.57,A -85,B 0,C 180,E1 -2174.193,E2 -2174.193} C_VEL
LIN {X 0,Y 573.257,Z 134.58,A -85,B 0,C 180,E1 -2177.112,E2 -2177.112} C_VEL
LIN {X 0,Y 573.248,Z 134.571,A -85,B 0,C 180,E1 -2180.077,E2 -2180.077} C_VEL
LIN {X 0,Y 573.232,Z 134.583,A -85,B 0,C 180,E1 -2183.1,E2 -2183.1} C_VEL
LIN {X 0,Y 573.254,Z 134.573,A -85,B 0,C 180,E1 -2185.41,E2 -2185.41} C_VEL
LIN {X 0,Y 573.249,Z 134.571,A -85,B 0,C 180,E1 -2188.029,E2 -2188.029} C_VEL
LIN {X 0,Y 573.237,Z 134.583,A -85,B 0,C 180,E1 -2190.884,E2 -2190.884} C_VEL
LIN {X 0,Y 573.261,Z 134.57,A -85,B 0,C 180,E1 -2193.525,E2 -2193.525} C_VEL
LIN {X 0,Y 573.214,Z 134.578,A -85,B 0,C 180,E1 -2196.052,E2 -2196.052} C_VEL
LIN {X 0,Y 573.24,Z 134.581,A -85,B 0,C 180,E1 -2198.702,E2 -2198.702} C_VEL
LIN {X 0,Y 573.229,Z 134.576,A -85,B 0,C 180,E1 -2201.593,E2 -2201.593} C_VEL
LIN {X 0,Y 573.232,Z 134.583,A -85,B 0,C 180,E1 -2204.334,E2 -2204.334} C_VEL
LIN {X 0,Y 573.239,Z 134.574,A -85,B 0,C 180,E1 -2207.359,E2 -2207.359} C_VEL
LIN {X 0,Y 573.253,Z 134.578,A -85,B 0,C 180,E1 -2210.568,E2 -2210.568} C_VEL
LIN {X 0,Y 573.253,Z 134.573,A -85,B 0,C 180,E1 -2213.078,E2 -2213.078} C_VEL
LIN {X 0,Y 573.267,Z 134.573,A -85,B 0,C 180,E1 -2215.672,E2 -2215.672} C_VEL
LIN {X 0,Y 573.248,Z 134.582,A -85,B 0,C 180,E1 -2218.185,E2 -2218.185} C_VEL
LIN {X 0,Y 573.262,Z 134.574,A -85,B 0,C 180,E1 -2220.634,E2 -2220.634} C_VEL
LIN {X 0,Y 573.252,Z 134.576,A -85,B 0,C 180,E1 -2223.024,E2 -2223.024} C_VEL
LIN {X 0,Y 573.292,Z 134.723,A -85,B 0,C 180,E1 -2225.141,E2 -2225.141} C_VEL
LIN {X 0,Y 573.819,Z 138.989,A -85,B 0,C 180,E1 -2225.969,E2 -2225.969} C_VEL
LIN {X 0,Y 573.606,Z 155.115,A -85,B 0,C 180,E1 -2228.902,E2 -2228.902} C_VEL
LIN {X 0,Y 573.482,Z 169.253,A -85,B 0,C 180,E1 -2231.42,E2 -2231.42} C_VEL
LIN {X 0,Y 573.39,Z 185.855,A -85,B 0,C 180,E1 -2234.357,E2 -2234.357} C_VEL
LIN {X 0,Y 573.308,Z 196.258,A -85,B 0,C 180,E1 -2236.147,E2 -2236.147} C_VEL
LIN {X 0,Y 573.622,Z 198.437,A -85,B 0,C 180,E1 -2236.219,E2 -2236.219} C_VEL
LIN {X 0,Y 574.047,Z 204.097,A -85,B 0,C 180,E1 -2236.301,E2 -2236.301} C_VEL
LIN {X 0,Y 573.888,Z 302.616,A -85,B 0,C 180,E1 -2237.558,E2 -2237.558} C_VEL
LIN {X 0,Y 573.816,Z 313.741,A -85,B 0,C 180,E1 -2237.803,E2 -2237.803} C_VEL
LIN {X 0,Y 573.725,Z 326.17,A -85,B 0,C 180,E1 -2238.205,E2 -2238.205} C_VEL
LIN {X 0,Y 573.619,Z 338.109,A -85,B 0,C 180,E1 -2238.742,E2 -2238.742} C_VEL
LIN {X 0,Y 573.495,Z 348.153,A -85,B 0,C 180,E1 -2239.319,E2 -2239.319} C_VEL
LIN {X 0,Y 573.395,Z 358.185,A -85,B 0,C 180,E1 -2240.03,E2 -2240.03} C_VEL
LIN {X 0,Y 573.32,Z 365.551,A -85,B 0,C 180,E1 -2240.652,E2 -2240.652} C_VEL
LIN {X 0,Y 573.197,Z 372.738,A -85,B 0,C 180,E1 -2241.362,E2 -2241.362} C_VEL
LIN {X 0,Y 573.16,Z 380.284,A -85,B 0,C 180,E1 -2242.248,E2 -2242.248} C_VEL
LIN {X 0,Y 573.07,Z 386.559,A -85,B 0,C 180,E1 -2243.13,E2 -2243.13} C_VEL
LIN {X 0,Y 573.074,Z 391.809,A -85,B 0,C 180,E1 -2244.017,E2 -2244.017} C_VEL
LIN {X 0,Y 572.962,Z 396.906,A -85,B 0,C 180,E1 -2245.074,E2 -2245.074} C_VEL
LIN {X 0,Y 573.015,Z 400.86,A -85,B 0,C 180,E1 -2246.132,E2 -2246.132} C_VEL
LIN {X 0,Y 572.959,Z 403.779,A -85,B 0,C 180,E1 -2247.188,E2 -2247.188} C_VEL
LIN {X 0,Y 572.946,Z 406.194,A -85,B 0,C 180,E1 -2248.594,E2 -2248.594} C_VEL
LIN {X 0,Y 572.941,Z 406.781,A -85,B 0,C 180,E1 -2249.297,E2 -2249.297} C_VEL
LIN {X 0,Y 572.941,Z 406.781,A -85,B 0,C 180,E1 -2250.703,E2 -2250.703} C_VEL
LIN {X 0,Y 572.946,Z 406.194,A -85,B 0,C 180,E1 -2251.406,E2 -2251.406} C_VEL
LIN {X 0,Y 572.959,Z 403.779,A -85,B 0,C 180,E1 -2252.812,E2 -2252.812} C_VEL
LIN {X 0,Y 573.015,Z 400.86,A -85,B 0,C 180,E1 -2253.868,E2 -2253.868} C_VEL
LIN {X 0,Y 572.962,Z 396.906,A -85,B 0,C 180,E1 -2254.926,E2 -2254.926} C_VEL
LIN {X 0,Y 573.074,Z 391.809,A -85,B 0,C 180,E1 -2255.983,E2 -2255.983} C_VEL
LIN {X 0,Y 573.082,Z 385.425,A -85,B 0,C 180,E1 -2257.044,E2 -2257.044} C_VEL
LIN {X 0,Y 573.177,Z 377.5,A -85,B 0,C 180,E1 -2258.106,E2 -2258.106} C_VEL
LIN {X 0,Y 573.279,Z 369.358,A -85,B 0,C 180,E1 -2258.992,E2 -2258.992} C_VEL
LIN {X 0,Y 573.34,Z 359.317,A -85,B 0,C 180,E1 -2259.881,E2 -2259.881} C_VEL
LIN {X 0,Y 573.453,Z 350.836,A -85,B 0,C 180,E1 -2260.504,E2 -2260.504} C_VEL
LIN {X 0,Y 573.565,Z 340.648,A -85,B 0,C 180,E1 -2261.12,E2 -2261.12} C_VEL
LIN {X 0,Y 573.677,Z 330.502,A -85,B 0,C 180,E1 -2261.612,E2 -2261.612} C_VEL
LIN {X 0,Y 573.796,Z 319.767,A -85,B 0,C 180,E1 -2262.018,E2 -2262.018} C_VEL
LIN {X 0,Y 573.859,Z 306.437,A -85,B 0,C 180,E1 -2262.376,E2 -2262.376} C_VEL
LIN {X 0,Y 573.936,Z 288.165,A -85,B 0,C 180,E1 -2262.643,E2 -2262.643} C_VEL
LIN {X 0,Y 573.942,Z 200.42,A -85,B 0,C 180,E1 -2263.748,E2 -2263.748} C_VEL
LIN {X 0,Y 573.346,Z 196.582,A -85,B 0,C 180,E1 -2263.829,E2 -2263.829} C_VEL
LIN {X 0,Y 573.295,Z 195.168,A -85,B 0,C 180,E1 -2264.011,E2 -2264.011} C_VEL
LIN {X 0,Y 573.388,Z 179.798,A -85,B 0,C 180,E1 -2266.714,E2 -2266.714} C_VEL
LIN {X 0,Y 573.544,Z 166.118,A -85,B 0,C 180,E1 -2269.134,E2 -2269.134} C_VEL
LIN {X 0,Y 573.649,Z 150.444,A -85,B 0,C 180,E1 -2271.942,E2 -2271.942} C_VEL
LIN {X 0,Y 573.801,Z 137.967,A -85,B 0,C 180,E1 -2274.224,E2 -2274.224} C_VEL
LIN {X 0,Y 573.277,Z 134.659,A -85,B 0,C 180,E1 -2274.879,E2 -2274.879} C_VEL
LIN {X 0,Y 573.274,Z 134.578,A -85,B 0,C 180,E1 -2277.765,E2 -2277.765} C_VEL
LIN {X 0,Y 573.25,Z 134.581,A -85,B 0,C 180,E1 -2280.176,E2 -2280.176} C_VEL
LIN {X 0,Y 573.255,Z 134.573,A -85,B 0,C 180,E1 -2282.645,E2 -2282.645} C_VEL
LIN {X 0,Y 573.208,Z 134.579,A -85,B 0,C 180,E1 -2285.187,E2 -2285.187} C_VEL
LIN {X 0,Y 573.237,Z 134.584,A -85,B 0,C 180,E1 -2287.807,E2 -2287.807} C_VEL
LIN {X 0,Y 573.245,Z 134.571,A -85,B 0,C 180,E1 -2290.525,E2 -2290.525} C_VEL
LIN {X 0,Y 573.236,Z 134.581,A -85,B 0,C 180,E1 -2293.359,E2 -2293.359} C_VEL
LIN {X 0,Y 573.244,Z 134.574,A -85,B 0,C 180,E1 -2296.331,E2 -2296.331} C_VEL
LIN {X 0,Y 573.229,Z 134.576,A -85,B 0,C 180,E1 -2298.542,E2 -2298.542} C_VEL
LIN {X 0,Y 573.24,Z 134.581,A -85,B 0,C 180,E1 -2301.298,E2 -2301.298} C_VEL
LIN {X 0,Y 573.213,Z 134.578,A -85,B 0,C 180,E1 -2304.018,E2 -2304.018} C_VEL
LIN {X 0,Y 573.284,Z 134.567,A -85,B 0,C 180,E1 -2306.518,E2 -2306.518} C_VEL
LIN {X 0,Y 573.237,Z 134.583,A -85,B 0,C 180,E1 -2309.116,E2 -2309.116} C_VEL
LIN {X 0,Y 573.249,Z 134.571,A -85,B 0,C 180,E1 -2311.971,E2 -2311.971} C_VEL
LIN {X 0,Y 573.254,Z 134.573,A -85,B 0,C 180,E1 -2314.59,E2 -2314.59} C_VEL
LIN {X 0,Y 573.233,Z 134.576,A -85,B 0,C 180,E1 -2317.662,E2 -2317.662} C_VEL
LIN {X 0,Y 573.276,Z 134.575,A -85,B 0,C 180,E1 -2320.728,E2 -2320.728} C_VEL
LIN {X 0,Y 573.246,Z 134.573,A -85,B 0,C 180,E1 -2323.621,E2 -2323.621} C_VEL
LIN {X 0,Y 573.271,Z 134.57,A -85,B 0,C 180,E1 -2325.807,E2 -2325.807} C_VEL
LIN {X 0,Y 573.259,Z 134.577,A -85,B 0,C 180,E1 -2328.745,E2 -2328.745} C_VEL
LIN {X 0,Y 573.281,Z 134.566,A -85,B 0,C 180,E1 -2331.54,E2 -2331.54} C_VEL
LIN {X 0,Y 573.287,Z 134.575,A -85,B 0,C 180,E1 -2334.371,E2 -2334.371} C_VEL
LIN {X 0,Y 573.305,Z 134.567,A -85,B 0,C 180,E1 -2337.892,E2 -2337.892} C_VEL
LIN {X 0,Y 573.329,Z 134.565,A -85,B 0,C 180,E1 -2340.702,E2 -2340.702} C_VEL
LIN {X 0,Y 573.235,Z 134.575,A -85,B 0,C 180,E1 -2343.514,E2 -2343.514} C_VEL
LIN {X 0,Y 573.289,Z 134.57,A -85,B 0,C 180,E1 -2345.628,E2 -2345.628} C_VEL
LIN {X 0,Y 573.281,Z 134.571,A -85,B 0,C 180,E1 -2348.459,E2 -2348.459} C_VEL
LIN {X 0,Y 573.267,Z 134.569,A -85,B 0,C 180,E1 -2351.312,E2 -2351.312} C_VEL
LIN {X 0,Y 573.27,Z 134.577,A -85,B 0,C 180,E1 -2354.193,E2 -2354.193} C_VEL
LIN {X 0,Y 573.255,Z 134.572,A -85,B 0,C 180,E1 -2357.111,E2 -2357.111} C_VEL
LIN {X 0,Y 573.247,Z 134.578,A -85,B 0,C 180,E1 -2360.076,E2 -2360.076} C_VEL
LIN {X 0,Y 573.229,Z 134.577,A -85,B 0,C 180,E1 -2363.099,E2 -2363.099} C_VEL
LIN {X 0,Y 573.245,Z 134.575,A -85,B 0,C 180,E1 -2364.381,E2 -2364.381} C_VEL
LIN {X 0,Y 572.619,Z 134.653,A -85,B 0,C 180,E1 -2364.968,E2 -2364.968} C_VEL
LIN {X 0,Y 569.782,Z 135.009,A -85,B 0,C 180,E1 -2365.92,E2 -2365.92} C_VEL
LIN {X 0,Y 567.354,Z 135.312,A -85,B 0,C 180,E1 -2366.685,E2 -2366.685} C_VEL
LIN {X 0,Y 566.302,Z 135.44,A -85,B 0,C 180,E1 -2367.277,E2 -2367.277} C_VEL
LIN {X 0,Y 566.213,Z 135.45,A -85,B 0,C 180,E1 -2367.477,E2 -2367.477} C_VEL
LIN {X 0,Y 566.182,Z 135.454,A -85,B 0,C 180,E1 -2370.592,E2 -2370.592} C_VEL
LIN {X 0,Y 566.224,Z 135.452,A -85,B 0,C 180,E1 -2373.101,E2 -2373.101} C_VEL
LIN {X 0,Y 566.207,Z 135.456,A -85,B 0,C 180,E1 -2375.688,E2 -2375.688} C_VEL
LIN {X 0,Y 566.21,Z 135.451,A -85,B 0,C 180,E1 -2378.559,E2 -2378.559} C_VEL
LIN {X 0,Y 566.207,Z 135.456,A -85,B 0,C 180,E1 -2381.136,E2 -2381.136} C_VEL
LIN {X 0,Y 566.196,Z 135.452,A -85,B 0,C 180,E1 -2384.035,E2 -2384.035} C_VEL
LIN {X 0,Y 566.197,Z 135.455,A -85,B 0,C 180,E1 -2387.083,E2 -2387.083} C_VEL
LIN {X 0,Y 566.222,Z 135.448,A -85,B 0,C 180,E1 -2389.803,E2 -2389.803} C_VEL
LIN {X 0,Y 566.195,Z 135.456,A -85,B 0,C 180,E1 -2392.599,E2 -2392.599} C_VEL
LIN {X 0,Y 566.215,Z 135.452,A -85,B 0,C 180,E1 -2395.183,E2 -2395.183} C_VEL
LIN {X 0,Y 566.23,Z 135.448,A -85,B 0,C 180,E1 -2397.744,E2 -2397.744} C_VEL
LIN {X 0,Y 566.224,Z 135.45,A -85,B 0,C 180,E1 -2400.323,E2 -2400.323} C_VEL
LIN {X 0,Y 566.208,Z 135.459,A -85,B 0,C 180,E1 -2402.661,E2 -2402.661} C_VEL
LIN {X 0,Y 566.232,Z 135.452,A -85,B 0,C 180,E1 -2405.039,E2 -2405.039} C_VEL
LIN {X 0,Y 566.192,Z 135.456,A -85,B 0,C 180,E1 -2408.138,E2 -2408.138} C_VEL
LIN {X 0,Y 566.233,Z 135.456,A -85,B 0,C 180,E1 -2410.612,E2 -2410.612} C_VEL
LIN {X 0,Y 566.213,Z 135.451,A -85,B 0,C 180,E1 -2413.412,E2 -2413.412} C_VEL
LIN {X 0,Y 566.195,Z 135.462,A -85,B 0,C 180,E1 -2416.359,E2 -2416.359} C_VEL
LIN {X 0,Y 566.231,Z 135.452,A -85,B 0,C 180,E1 -2418.675,E2 -2418.675} C_VEL
LIN {X 0,Y 566.231,Z 135.449,A -85,B 0,C 180,E1 -2421.434,E2 -2421.434} C_VEL
LIN {X 0,Y 566.259,Z 135.452,A -85,B 0,C 180,E1 -2424.302,E2 -2424.302} C_VEL
LIN {X 0,Y 566.283,Z 135.449,A -85,B 0,C 180,E1 -2427.866,E2 -2427.866} C_VEL
LIN {X 0,Y 566.3,Z 135.441,A -85,B 0,C 180,E1 -2430.711,E2 -2430.711} C_VEL
LIN {X 0,Y 566.269,Z 135.444,A -85,B 0,C 180,E1 -2432.846,E2 -2432.846} C_VEL
LIN {X 0,Y 566.259,Z 135.452,A -85,B 0,C 180,E1 -2435.698,E2 -2435.698} C_VEL
LIN {X 0,Y 566.231,Z 135.449,A -85,B 0,C 180,E1 -2438.566,E2 -2438.566} C_VEL
LIN {X 0,Y 566.239,Z 135.453,A -85,B 0,C 180,E1 -2441.454,E2 -2441.454} C_VEL
LIN {X 0,Y 566.231,Z 135.449,A -85,B 0,C 180,E1 -2444.507,E2 -2444.507} C_VEL
LIN {X 0,Y 566.197,Z 135.459,A -85,B 0,C 180,E1 -2447.332,E2 -2447.332} C_VEL
LIN {X 0,Y 566.211,Z 135.451,A -85,B 0,C 180,E1 -2450.337,E2 -2450.337} C_VEL
LIN {X 0,Y 566.186,Z 135.463,A -85,B 0,C 180,E1 -2453.404,E2 -2453.404} C_VEL
LIN {X 0,Y 566.21,Z 135.454,A -85,B 0,C 180,E1 -2455.749,E2 -2455.749} C_VEL
LIN {X 0,Y 566.202,Z 135.451,A -85,B 0,C 180,E1 -2458.203,E2 -2458.203} C_VEL
LIN {X 0,Y 566.19,Z 135.453,A -85,B 0,C 180,E1 -2460.592,E2 -2460.592} C_VEL
LIN {X 0,Y 566.225,Z 135.456,A -85,B 0,C 180,E1 -2463.101,E2 -2463.101} C_VEL
LIN {X 0,Y 566.202,Z 135.45,A -85,B 0,C 180,E1 -2466.215,E2 -2466.215} C_VEL
LIN {X 0,Y 566.219,Z 135.452,A -85,B 0,C 180,E1 -2469.273,E2 -2469.273} C_VEL
LIN {X 0,Y 566.206,Z 135.444,A -85,B 0,C 180,E1 -2472.088,E2 -2472.088} C_VEL
LIN {X 0,Y 566.169,Z 135.461,A -85,B 0,C 180,E1 -2475.036,E2 -2475.036} C_VEL
LIN {X 0,Y 566.212,Z 135.45,A -85,B 0,C 180,E1 -2477.913,E2 -2477.913} C_VEL
LIN {X 0,Y 566.216,Z 135.458,A -85,B 0,C 180,E1 -2480.727,E2 -2480.727} C_VEL
LIN {X 0,Y 566.213,Z 135.45,A -85,B 0,C 180,E1 -2483.783,E2 -2483.783} C_VEL
LIN {X 0,Y 566.224,Z 135.451,A -85,B 0,C 180,E1 -2486.263,E2 -2486.263} C_VEL
LIN {X 0,Y 566.194,Z 135.455,A -85,B 0,C 180,E1 -2488.922,E2 -2488.922} C_VEL
LIN {X 0,Y 566.223,Z 135.449,A -85,B 0,C 180,E1 -2491.859,E2 -2491.859} C_VEL
LIN {X 0,Y 566.221,Z 135.455,A -85,B 0,C 180,E1 -2494.252,E2 -2494.252} C_VEL
LIN {X 0,Y 566.187,Z 135.456,A -85,B 0,C 180,E1 -2496.714,E2 -2496.714} C_VEL
LIN {X 0,Y 566.208,Z 135.451,A -85,B 0,C 180,E1 -2499.663,E2 -2499.663} C_VEL
LIN {X 0,Y 566.199,Z 135.452,A -85,B 0,C 180,E1 -2502.669,E2 -2502.669} C_VEL
LIN {X 0,Y 566.23,Z 135.452,A -85,B 0,C 180,E1 -2505.627,E2 -2505.627} C_VEL
LIN {X 0,Y 566.23,Z 135.445,A -85,B 0,C 180,E1 -2508.676,E2 -2508.676} C_VEL
LIN {X 0,Y 566.225,Z 135.448,A -85,B 0,C 180,E1 -2511.435,E2 -2511.435} C_VEL
LIN {X 0,Y 566.257,Z 135.446,A -85,B 0,C 180,E1 -2514.302,E2 -2514.302} C_VEL
LIN {X 0,Y 566.276,Z 135.445,A -85,B 0,C 180,E1 -2517.867,E2 -2517.867} C_VEL
LIN {X 0,Y 566.299,Z 135.435,A -85,B 0,C 180,E1 -2520.711,E2 -2520.711} C_VEL
LIN {X 0,Y 566.27,Z 135.442,A -85,B 0,C 180,E1 -2522.846,E2 -2522.846} C_VEL
LIN {X 0,Y 566.256,Z 135.45,A -85,B 0,C 180,E1 -2525.699,E2 -2525.699} C_VEL
LIN {X 0,Y 566.225,Z 135.445,A -85,B 0,C 180,E1 -2528.566,E2 -2528.566} C_VEL
LIN {X 0,Y 566.239,Z 135.453,A -85,B 0,C 180,E1 -2531.455,E2 -2531.455} C_VEL
LIN {X 0,Y 566.232,Z 135.448,A -85,B 0,C 180,E1 -2534.507,E2 -2534.507} C_VEL
LIN {X 0,Y 566.2,Z 135.454,A -85,B 0,C 180,E1 -2537.332,E2 -2537.332} C_VEL
LIN {X 0,Y 566.21,Z 135.448,A -85,B 0,C 180,E1 -2540.338,E2 -2540.338} C_VEL
LIN {X 0,Y 566.171,Z 135.46,A -85,B 0,C 180,E1 -2543.282,E2 -2543.282} C_VEL
LIN {X 0,Y 566.213,Z 135.447,A -85,B 0,C 180,E1 -2545.749,E2 -2545.749} C_VEL
LIN {X 0,Y 566.2,Z 135.45,A -85,B 0,C 180,E1 -2548.203,E2 -2548.203} C_VEL
LIN {X 0,Y 566.197,Z 135.457,A -85,B 0,C 180,E1 -2551.078,E2 -2551.078} C_VEL
LIN {X 0,Y 566.211,Z 135.447,A -85,B 0,C 180,E1 -2553.735,E2 -2553.735} C_VEL
LIN {X 0,Y 566.199,Z 135.459,A -85,B 0,C 180,E1 -2556.57,E2 -2556.57} C_VEL
LIN {X 0,Y 566.214,Z 135.448,A -85,B 0,C 180,E1 -2559.686,E2 -2559.686} C_VEL
LIN {X 0,Y 566.201,Z 135.454,A -85,B 0,C 180,E1 -2562.918,E2 -2562.918} C_VEL
LIN {X 0,Y 566.194,Z 135.456,A -85,B 0,C 180,E1 -2566.05,E2 -2566.05} C_VEL
LIN {X 0,Y 566.204,Z 135.448,A -85,B 0,C 180,E1 -2569.215,E2 -2569.215} C_VEL
LIN {X 0,Y 566.19,Z 135.454,A -85,B 0,C 180,E1 -2571.638,E2 -2571.638} C_VEL
LIN {X 0,Y 566.164,Z 135.462,A -85,B 0,C 180,E1 -2574.308,E2 -2574.308} C_VEL
LIN {X 0,Y 566.221,Z 135.449,A -85,B 0,C 180,E1 -2576.898,E2 -2576.898} C_VEL
LIN {X 0,Y 566.188,Z 135.456,A -85,B 0,C 180,E1 -2579.408,E2 -2579.408} C_VEL
LIN {X 0,Y 566.214,Z 135.459,A -85,B 0,C 180,E1 -2581.858,E2 -2581.858} C_VEL
LIN {X 0,Y 566.252,Z 135.501,A -85,B 0,C 180,E1 -2584.952,E2 -2584.952} C_VEL
LIN {X 0,Y 566.869,Z 139.941,A -85,B 0,C 180,E1 -2585.85,E2 -2585.85} C_VEL
LIN {X 0,Y 566.606,Z 156.571,A -85,B 0,C 180,E1 -2588.918,E2 -2588.918} C_VEL
LIN {X 0,Y 566.472,Z 170.167,A -85,B 0,C 180,E1 -2591.369,E2 -2591.369} C_VEL
LIN {X 0,Y 566.338,Z 185.831,A -85,B 0,C 180,E1 -2594.157,E2 -2594.157} C_VEL
LIN {X 0,Y 566.28,Z 196.267,A -85,B 0,C 180,E1 -2595.972,E2 -2595.972} C_VEL
LIN {X 0,Y 566.608,Z 198.437,A -85,B 0,C 180,E1 -2596.045,E2 -2596.045} C_VEL
LIN {X 0,Y 567.155,Z 204.097,A -85,B 0,C 180,E1 -2596.131,E2 -2596.131} C_VEL
LIN {X 0,Y 566.965,Z 302.549,A -85,B 0,C 180,E1 -2597.403,E2 -2597.403} C_VEL
LIN {X 0,Y 566.895,Z 313.701,A -85,B 0,C 180,E1 -2597.652,E2 -2597.652} C_VEL
LIN {X 0,Y 566.761,Z 326.166,A -85,B 0,C 180,E1 -2598.058,E2 -2598.058} C_VEL
LIN {X 0,Y 566.628,Z 339.026,A -85,B 0,C 180,E1 -2598.653,E2 -2598.653} C_VEL
LIN {X 0,Y 566.474,Z 349.468,A -85,B 0,C 180,E1 -2599.275,E2 -2599.275} C_VEL
LIN {X 0,Y 566.39,Z 358.169,A -85,B 0,C 180,E1 -2599.906,E2 -2599.906} C_VEL
LIN {X 0,Y 566.303,Z 365.538,A -85,B 0,C 180,E1 -2600.536,E2 -2600.536} C_VEL
LIN {X 0,Y 566.159,Z 372.728,A -85,B 0,C 180,E1 -2601.253,E2 -2601.253} C_VEL
LIN {X 0,Y 566.094,Z 380.274,A -85,B 0,C 180,E1 -2602.151,E2 -2602.151} C_VEL
LIN {X 0,Y 566.004,Z 386.679,A -85,B 0,C 180,E1 -2603.064,E2 -2603.064} C_VEL
LIN {X 0,Y 565.989,Z 391.798,A -85,B 0,C 180,E1 -2603.941,E2 -2603.941} C_VEL
LIN {X 0,Y 565.877,Z 396.896,A -85,B 0,C 180,E1 -2605.013,E2 -2605.013} C_VEL
LIN {X 0,Y 565.926,Z 400.852,A -85,B 0,C 180,E1 -2606.084,E2 -2606.084} C_VEL
LIN {X 0,Y 565.878,Z 403.773,A -85,B 0,C 180,E1 -2607.152,E2 -2607.152} C_VEL
LIN {X 0,Y 565.846,Z 406.196,A -85,B 0,C 180,E1 -2608.577,E2 -2608.577} C_VEL
LIN {X 0,Y 565.841,Z 406.78,A -85,B 0,C 180,E1 -2609.288,E2 -2609.288} C_VEL
LIN {X 0,Y 565.841,Z 406.78,A -85,B 0,C 180,E1 -2610.712,E2 -2610.712} C_VEL
LIN {X 0,Y 565.846,Z 406.196,A -85,B 0,C 180,E1 -2611.423,E2 -2611.423} C_VEL
LIN {X 0,Y 565.878,Z 403.773,A -85,B 0,C 180,E1 -2612.848,E2 -2612.848} C_VEL
LIN {X 0,Y 565.926,Z 400.852,A -85,B 0,C 180,E1 -2613.916,E2 -2613.916} C_VEL
LIN {X 0,Y 565.877,Z 396.896,A -85,B 0,C 180,E1 -2614.987,E2 -2614.987} C_VEL
LIN {X 0,Y 565.99,Z 391.798,A -85,B 0,C 180,E1 -2616.059,E2 -2616.059} C_VEL
LIN {X 0,Y 566.004,Z 386.679,A -85,B 0,C 180,E1 -2616.936,E2 -2616.936} C_VEL
LIN {X 0,Y 566.094,Z 380.274,A -85,B 0,C 180,E1 -2617.849,E2 -2617.849} C_VEL
LIN {X 0,Y 566.159,Z 372.728,A -85,B 0,C 180,E1 -2618.747,E2 -2618.747} C_VEL
LIN {X 0,Y 566.296,Z 363.619,A -85,B 0,C 180,E1 -2619.645,E2 -2619.645} C_VEL
LIN {X 0,Y 566.434,Z 352.166,A -85,B 0,C 180,E1 -2620.545,E2 -2620.545} C_VEL
LIN {X 0,Y 566.56,Z 342.766,A -85,B 0,C 180,E1 -2621.14,E2 -2621.14} C_VEL
LIN {X 0,Y 566.701,Z 332.689,A -85,B 0,C 180,E1 -2621.658,E2 -2621.658} C_VEL
LIN {X 0,Y 566.795,Z 322.318,A -85,B 0,C 180,E1 -2622.078,E2 -2622.078} C_VEL
LIN {X 0,Y 566.911,Z 311.954,A -85,B 0,C 180,E1 -2622.393,E2 -2622.393} C_VEL
LIN {X 0,Y 566.961,Z 301.218,A -85,B 0,C 180,E1 -2622.62,E2 -2622.62} C_VEL
LIN {X 0,Y 567.075,Z 201.315,A -85,B 0,C 180,E1 -2623.906,E2 -2623.906} C_VEL
LIN {X 0,Y 566.319,Z 196.597,A -85,B 0,C 180,E1 -2624.004,E2 -2624.004} C_VEL
LIN {X 0,Y 566.267,Z 195.168,A -85,B 0,C 180,E1 -2624.189,E2 -2624.189} C_VEL
LIN {X 0,Y 566.366,Z 180.011,A -85,B 0,C 180,E1 -2626.875,E2 -2626.875} C_VEL
LIN {X 0,Y 566.56,Z 165.43,A -85,B 0,C 180,E1 -2629.48,E2 -2629.48} C_VEL
LIN {X 0,Y 566.72,Z 148.278,A -85,B 0,C 180,E1 -2632.609,E2 -2632.609} C_VEL
LIN {X 0,Y 566.827,Z 138.92,A -85,B 0,C 180,E1 -2634.347,E2 -2634.347} C_VEL
LIN {X 0,Y 566.238,Z 135.519,A -85,B 0,C 180,E1 -2635.033,E2 -2635.033} C_VEL
